LIN {X 0,Y 383.018,Z 410.271,A -85,B 0,C 180,E1 -11844.045,E2 -11844.045} C_VEL
LIN {X 0,Y 382.98,Z 410.277,A -85,B 0,C 180,E1 -11847.578,E2 -11847.578} C_VEL
LIN {X 0,Y 382.99,Z 410.275,A -85,B 0,C 180,E1 -11850.301,E2 -11850.301} C_VEL
LIN {X 0,Y 383.048,Z 410.271,A -85,B 0,C 180,E1 -11852.698,E2 -11852.698} C_VEL
LIN {X 0,Y 383.043,Z 410.273,A -85,B 0,C 180,E1 -11855.04,E2 -11855.04} C_VEL
LIN {X 0,Y 382.984,Z 410.277,A -85,B 0,C 180,E1 -11858.469,E2 -11858.469} C_VEL
LIN {X 0,Y 383.054,Z 410.266,A -85,B 0,C 180,E1 -11861.827,E2 -11861.827} C_VEL
LIN {X 0,Y 383.102,Z 410.263,A -85,B 0,C 180,E1 -11865.119,E2 -11865.119} C_VEL
LIN {X 0,Y 383.089,Z 410.265,A -85,B 0,C 180,E1 -11868.358,E2 -11868.358} C_VEL
LIN {X 0,Y 383.256,Z 410.242,A -85,B 0,C 180,E1 -11871.976,E2 -11871.976} C_VEL
LIN {X 0,Y 383.192,Z 410.255,A -85,B 0,C 180,E1 -11874.739,E2 -11874.739} C_VEL
LIN {X 0,Y 383.38,Z 410.227,A -85,B 0,C 180,E1 -11877.899,E2 -11877.899} C_VEL
LIN {X 0,Y 383.511,Z 410.211,A -85,B 0,C 180,E1 -11880.001,E2 -11880.001} C_VEL
LIN {X 0,Y 383.245,Z 410.243,A -85,B 0,C 180,E1 -11883.154,E2 -11883.154} C_VEL
LIN {X 0,Y 383.276,Z 410.244,A -85,B 0,C 180,E1 -11886.317,E2 -11886.317} C_VEL
LIN {X 0,Y 383.144,Z 410.255,A -85,B 0,C 180,E1 -11889.503,E2 -11889.503} C_VEL
LIN {X 0,Y 383.119,Z 410.259,A -85,B 0,C 180,E1 -11893.537,E2 -11893.537} C_VEL
LIN {X 0,Y 383.09,Z 410.262,A -85,B 0,C 180,E1 -11897.456,E2 -11897.456} C_VEL
LIN {X 0,Y 383.022,Z 410.272,A -85,B 0,C 180,E1 -11900.648,E2 -11900.648} C_VEL
LIN {X 0,Y 383.02,Z 410.274,A -85,B 0,C 180,E1 -11903.809,E2 -11903.809} C_VEL
LIN {X 0,Y 383.075,Z 410.271,A -85,B 0,C 180,E1 -11906.124,E2 -11906.124} C_VEL
LIN {X 0,Y 383.045,Z 410.27,A -85,B 0,C 180,E1 -11908.493,E2 -11908.493} C_VEL
LIN {X 0,Y 383.004,Z 410.275,A -85,B 0,C 180,E1 -11912.428,E2 -11912.428} C_VEL
LIN {X 0,Y 383.023,Z 410.277,A -85,B 0,C 180,E1 -11915.956,E2 -11915.956} C_VEL
LIN {X 0,Y 383.003,Z 410.279,A -85,B 0,C 180,E1 -11917.906,E2 -11917.906} C_VEL
LIN {X 0,Y 383.458,Z 413.122,A -85,B 0,C 180,E1 -11921.286,E2 -11921.286} C_VEL
LIN {X 0,Y 383.841,Z 416.038,A -85,B 0,C 180,E1 -11924.434,E2 -11924.434} C_VEL
LIN {X 0,Y 384.047,Z 419.017,A -85,B 0,C 180,E1 -11927.384,E2 -11927.384} C_VEL
LIN {X 0,Y 383.867,Z 422.184,A -85,B 0,C 180,E1 -11930.261,E2 -11930.261} C_VEL
LIN {X 0,Y 383.627,Z 425.155,A -85,B 0,C 180,E1 -11932.804,E2 -11932.804} C_VEL
LIN {X 0,Y 383.174,Z 429.849,A -85,B 0,C 180,E1 -11936.617,E2 -11936.617} C_VEL
LIN {X 0,Y 382.802,Z 433.782,A -85,B 0,C 180,E1 -11939.643,E2 -11939.643} C_VEL
LIN {X 0,Y 382.489,Z 437.86,A -85,B 0,C 180,E1 -11942.655,E2 -11942.655} C_VEL
LIN {X 0,Y 382.143,Z 442.74,A -85,B 0,C 180,E1 -11946.134,E2 -11946.134} C_VEL
LIN {X 0,Y 381.924,Z 448.017,A -85,B 0,C 180,E1 -11949.799,E2 -11949.799} C_VEL
LIN {X 0,Y 381.826,Z 450.081,A -85,B 0,C 180,E1 -11951.106,E2 -11951.106} C_VEL
LIN {X 0,Y 384.052,Z 460.663,A -85,B 0,C 180,E1 -11951.573,E2 -11951.573} C_VEL
LIN {X 0,Y 385.927,Z 471.661,A -85,B 0,C 180,E1 -11952.19,E2 -11952.19} C_VEL
LIN {X 0,Y 387.212,Z 482.447,A -85,B 0,C 180,E1 -11952.932,E2 -11952.932} C_VEL
LIN {X 0,Y 386.342,Z 494.597,A -85,B 0,C 180,E1 -11953.894,E2 -11953.894} C_VEL
LIN {X 0,Y 385.407,Z 504.894,A -85,B 0,C 180,E1 -11954.939,E2 -11954.939} C_VEL
LIN {X 0,Y 384.745,Z 512.361,A -85,B 0,C 180,E1 -11955.844,E2 -11955.844} C_VEL
LIN {X 0,Y 384.005,Z 520.647,A -85,B 0,C 180,E1 -11957.045,E2 -11957.045} C_VEL
LIN {X 0,Y 383.354,Z 526.848,A -85,B 0,C 180,E1 -11958.098,E2 -11958.098} C_VEL
LIN {X 0,Y 382.768,Z 533.386,A -85,B 0,C 180,E1 -11959.42,E2 -11959.42} C_VEL
LIN {X 0,Y 382.409,Z 537.889,A -85,B 0,C 180,E1 -11960.48,E2 -11960.48} C_VEL
LIN {X 0,Y 381.991,Z 543.381,A -85,B 0,C 180,E1 -11962.069,E2 -11962.069} C_VEL
LIN {X 0,Y 381.712,Z 547.705,A -85,B 0,C 180,E1 -11963.658,E2 -11963.658} C_VEL
LIN {X 0,Y 381.647,Z 550.072,A -85,B 0,C 180,E1 -11964.717,E2 -11964.717} C_VEL
LIN {X 0,Y 381.629,Z 551.872,A -85,B 0,C 180,E1 -11965.776,E2 -11965.776} C_VEL
LIN {X 0,Y 381.561,Z 554.315,A -85,B 0,C 180,E1 -11967.889,E2 -11967.889} C_VEL
LIN {X 0,Y 381.603,Z 554.905,A -85,B 0,C 180,E1 -11968.945,E2 -11968.945} C_VEL
LIN {X 0,Y 381.603,Z 554.905,A -85,B 0,C 180,E1 -11971.055,E2 -11971.055} C_VEL
LIN {X 0,Y 381.561,Z 554.315,A -85,B 0,C 180,E1 -11972.111,E2 -11972.111} C_VEL
LIN {X 0,Y 381.629,Z 551.872,A -85,B 0,C 180,E1 -11974.224,E2 -11974.224} C_VEL
LIN {X 0,Y 381.647,Z 550.072,A -85,B 0,C 180,E1 -11975.283,E2 -11975.283} C_VEL
LIN {X 0,Y 381.783,Z 546.464,A -85,B 0,C 180,E1 -11976.872,E2 -11976.872} C_VEL
LIN {X 0,Y 382.118,Z 541.721,A -85,B 0,C 180,E1 -11978.461,E2 -11978.461} C_VEL
LIN {X 0,Y 382.547,Z 535.697,A -85,B 0,C 180,E1 -11980.051,E2 -11980.051} C_VEL
LIN {X 0,Y 383.08,Z 529.6,A -85,B 0,C 180,E1 -11981.374,E2 -11981.374} C_VEL
LIN {X 0,Y 383.669,Z 523.9,A -85,B 0,C 180,E1 -11982.429,E2 -11982.429} C_VEL
LIN {X 0,Y 384.447,Z 515.345,A -85,B 0,C 180,E1 -11983.748,E2 -11983.748} C_VEL
LIN {X 0,Y 385.143,Z 507.162,A -85,B 0,C 180,E1 -11984.801,E2 -11984.801} C_VEL
LIN {X 0,Y 385.907,Z 498.65,A -85,B 0,C 180,E1 -11985.717,E2 -11985.717} C_VEL
LIN {X 0,Y 386.683,Z 489.935,A -85,B 0,C 180,E1 -11986.498,E2 -11986.498} C_VEL
LIN {X 0,Y 387.184,Z 482.448,A -85,B 0,C 180,E1 -11987.069,E2 -11987.069} C_VEL
LIN {X 0,Y 386.051,Z 472.502,A -85,B 0,C 180,E1 -11987.76,E2 -11987.76} C_VEL
LIN {X 0,Y 384.137,Z 461.226,A -85,B 0,C 180,E1 -11988.401,E2 -11988.401} C_VEL
LIN {X 0,Y 381.883,Z 450.583,A -85,B 0,C 180,E1 -11988.878,E2 -11988.878} C_VEL
LIN {X 0,Y 381.813,Z 449.839,A -85,B 0,C 180,E1 -11988.93,E2 -11988.93} C_VEL
LIN {X 0,Y 382.011,Z 445.986,A -85,B 0,C 180,E1 -11991.589,E2 -11991.589} C_VEL
LIN {X 0,Y 382.258,Z 441.065,A -85,B 0,C 180,E1 -11995.015,E2 -11995.015} C_VEL
LIN {X 0,Y 382.591,Z 436.226,A -85,B 0,C 180,E1 -11998.528,E2 -11998.528} C_VEL
LIN {X 0,Y 383.049,Z 431.432,A -85,B 0,C 180,E1 -12002.145,E2 -12002.145} C_VEL
LIN {X 0,Y 383.326,Z 428.263,A -85,B 0,C 180,E1 -12004.635,E2 -12004.635} C_VEL
LIN {X 0,Y 383.728,Z 424.136,A -85,B 0,C 180,E1 -12008.042,E2 -12008.042} C_VEL
LIN {X 0,Y 384,Z 420.345,A -85,B 0,C 180,E1 -12011.376,E2 -12011.376} C_VEL
LIN {X 0,Y 383.997,Z 417.514,A -85,B 0,C 180,E1 -12014.065,E2 -12014.065} C_VEL
LIN {X 0,Y 383.601,Z 414.374,A -85,B 0,C 180,E1 -12017.321,E2 -12017.321} C_VEL
LIN {X 0,Y 383.231,Z 411.685,A -85,B 0,C 180,E1 -12020.373,E2 -12020.373} C_VEL
LIN {X 0,Y 383.004,Z 410.279,A -85,B 0,C 180,E1 -12022.094,E2 -12022.094} C_VEL
LIN {X 0,Y 383.015,Z 410.279,A -85,B 0,C 180,E1 -12025.331,E2 -12025.331} C_VEL
LIN {X 0,Y 383.032,Z 410.274,A -85,B 0,C 180,E1 -12027.852,E2 -12027.852} C_VEL
LIN {X 0,Y 383.059,Z 410.27,A -85,B 0,C 180,E1 -12031.719,E2 -12031.719} C_VEL
LIN {X 0,Y 383.045,Z 410.268,A -85,B 0,C 180,E1 -12035.039,E2 -12035.039} C_VEL
LIN {X 0,Y 382.986,Z 410.276,A -85,B 0,C 180,E1 -12038.468,E2 -12038.468} C_VEL
LIN {X 0,Y 383.083,Z 410.269,A -85,B 0,C 180,E1 -12041.827,E2 -12041.827} C_VEL
LIN {X 0,Y 383.106,Z 410.261,A -85,B 0,C 180,E1 -12045.118,E2 -12045.118} C_VEL
LIN {X 0,Y 383.09,Z 410.263,A -85,B 0,C 180,E1 -12048.357,E2 -12048.357} C_VEL
LIN {X 0,Y 383.257,Z 410.244,A -85,B 0,C 180,E1 -12051.975,E2 -12051.975} C_VEL
LIN {X 0,Y 383.192,Z 410.249,A -85,B 0,C 180,E1 -12054.738,E2 -12054.738} C_VEL
LIN {X 0,Y 383.38,Z 410.228,A -85,B 0,C 180,E1 -12057.898,E2 -12057.898} C_VEL
LIN {X 0,Y 383.511,Z 410.211,A -85,B 0,C 180,E1 -12059.999,E2 -12059.999} C_VEL
LIN {X 0,Y 383.245,Z 410.246,A -85,B 0,C 180,E1 -12063.153,E2 -12063.153} C_VEL
LIN {X 0,Y 383.254,Z 410.242,A -85,B 0,C 180,E1 -12066.631,E2 -12066.631} C_VEL
LIN {X 0,Y 383.143,Z 410.26,A -85,B 0,C 180,E1 -12069.502,E2 -12069.502} C_VEL
LIN {X 0,Y 383.117,Z 410.262,A -85,B 0,C 180,E1 -12073.536,E2 -12073.536} C_VEL
LIN {X 0,Y 383.086,Z 410.266,A -85,B 0,C 180,E1 -12077.454,E2 -12077.454} C_VEL
LIN {X 0,Y 383.02,Z 410.272,A -85,B 0,C 180,E1 -12080.647,E2 -12080.647} C_VEL
LIN {X 0,Y 383.025,Z 410.271,A -85,B 0,C 180,E1 -12083.807,E2 -12083.807} C_VEL
LIN {X 0,Y 383.071,Z 410.264,A -85,B 0,C 180,E1 -12086.123,E2 -12086.123} C_VEL
LIN {X 0,Y 383.041,Z 410.27,A -85,B 0,C 180,E1 -12088.492,E2 -12088.492} C_VEL
LIN {X 0,Y 383.003,Z 410.273,A -85,B 0,C 180,E1 -12092.15,E2 -12092.15} C_VEL
LIN {X 0,Y 383.01,Z 410.276,A -85,B 0,C 180,E1 -12094.668,E2 -12094.668} C_VEL
LIN {X 0,Y 382.996,Z 410.274,A -85,B 0,C 180,E1 -12097.905,E2 -12097.905} C_VEL
LIN {X 0,Y 383.039,Z 410.27,A -85,B 0,C 180,E1 -12101.339,E2 -12101.339} C_VEL
LIN {X 0,Y 383.027,Z 410.272,A -85,B 0,C 180,E1 -12104.309,E2 -12104.309} C_VEL
LIN {X 0,Y 383.003,Z 410.274,A -85,B 0,C 180,E1 -12107.24,E2 -12107.24} C_VEL
LIN {X 0,Y 383.01,Z 410.276,A -85,B 0,C 180,E1 -12110.413,E2 -12110.413} C_VEL
LIN {X 0,Y 383.02,Z 410.272,A -85,B 0,C 180,E1 -12114.045,E2 -12114.045} C_VEL
LIN {X 0,Y 382.98,Z 410.276,A -85,B 0,C 180,E1 -12117.578,E2 -12117.578} C_VEL
LIN {X 0,Y 382.987,Z 410.279,A -85,B 0,C 180,E1 -12120.3,E2 -12120.3} C_VEL
LIN {X 0,Y 383.075,Z 410.266,A -85,B 0,C 180,E1 -12124.021,E2 -12124.021} C_VEL
LIN {X 0,Y 383.003,Z 410.273,A -85,B 0,C 180,E1 -12127.335,E2 -12127.335} C_VEL
LIN {X 0,Y 383.056,Z 410.272,A -85,B 0,C 180,E1 -12130.717,E2 -12130.717} C_VEL
LIN {X 0,Y 383.076,Z 410.27,A -85,B 0,C 180,E1 -12134.027,E2 -12134.027} C_VEL
LIN {X 0,Y 383.132,Z 410.26,A -85,B 0,C 180,E1 -12137.284,E2 -12137.284} C_VEL
LIN {X 0,Y 383.138,Z 410.274,A -85,B 0,C 180,E1 -12139.598,E2 -12139.598} C_VEL
LIN {X 0,Y 383.813,Z 412.56,A -85,B 0,C 180,E1 -12139.95,E2 -12139.95} C_VEL
LIN {X 0,Y 385.349,Z 414.562,A -85,B 0,C 180,E1 -12140.685,E2 -12140.685} C_VEL
LIN {X 0,Y 387.437,Z 415.864,A -85,B 0,C 180,E1 -12141.656,E2 -12141.656} C_VEL
LIN {X 0,Y 388.84,Z 416.565,A -85,B 0,C 180,E1 -12142.402,E2 -12142.402} C_VEL
LIN {X 0,Y 389.961,Z 418.835,A -85,B 0,C 180,E1 -12143.142,E2 -12143.142} C_VEL
LIN {X 0,Y 391.789,Z 420.997,A -85,B 0,C 180,E1 -12144.467,E2 -12144.467} C_VEL
LIN {X 0,Y 393.422,Z 422.062,A -85,B 0,C 180,E1 -12145.903,E2 -12145.903} C_VEL
LIN {X 0,Y 394.945,Z 422.432,A -85,B 0,C 180,E1 -12147.96,E2 -12147.96} C_VEL
LIN {X 0,Y 395.509,Z 422.495,A -85,B 0,C 180,E1 -12150,E2 -12150} C_VEL
LIN {X 0,Y 394.945,Z 422.432,A -85,B 0,C 180,E1 -12152.04,E2 -12152.04} C_VEL
LIN {X 0,Y 393.422,Z 422.062,A -85,B 0,C 180,E1 -12154.097,E2 -12154.097} C_VEL
LIN {X 0,Y 391.445,Z 420.702,A -85,B 0,C 180,E1 -12155.796,E2 -12155.796} C_VEL
LIN {X 0,Y 389.551,Z 418.156,A -85,B 0,C 180,E1 -12157.135,E2 -12157.135} C_VEL
LIN {X 0,Y 388.788,Z 416.4,A -85,B 0,C 180,E1 -12157.634,E2 -12157.634} C_VEL
LIN {X 0,Y 385.957,Z 415.055,A -85,B 0,C 180,E1 -12159.036,E2 -12159.036} C_VEL
LIN {X 0,Y 384.053,Z 412.977,A -85,B 0,C 180,E1 -12159.938,E2 -12159.938} C_VEL
LIN {X 0,Y 383.252,Z 410.915,A -85,B 0,C 180,E1 -12160.332,E2 -12160.332} C_VEL
LIN {X 0,Y 383.121,Z 410.262,A -85,B 0,C 180,E1 -12160.436,E2 -12160.436} C_VEL
LIN {X 0,Y 383.122,Z 410.265,A -85,B 0,C 180,E1 -12163.796,E2 -12163.796} C_VEL
LIN {X 0,Y 383.09,Z 410.267,A -85,B 0,C 180,E1 -12167.454,E2 -12167.454} C_VEL
LIN {X 0,Y 383.026,Z 410.27,A -85,B 0,C 180,E1 -12170.648,E2 -12170.648} C_VEL
LIN {X 0,Y 383.028,Z 410.274,A -85,B 0,C 180,E1 -12173.807,E2 -12173.807} C_VEL
LIN {X 0,Y 383.075,Z 410.265,A -85,B 0,C 180,E1 -12176.123,E2 -12176.123} C_VEL
LIN {X 0,Y 382.987,Z 410.279,A -85,B 0,C 180,E1 -12179.7,E2 -12179.7} C_VEL
LIN {X 0,Y 382.997,Z 410.28,A -85,B 0,C 180,E1 -12183.4,E2 -12183.4} C_VEL
LIN {X 0,Y 382.992,Z 410.272,A -85,B 0,C 180,E1 -12185.383,E2 -12185.383} C_VEL
LIN {X 0,Y 382.356,Z 410.354,A -85,B 0,C 180,E1 -12186.261,E2 -12186.261} C_VEL
LIN {X 0,Y 379.559,Z 410.706,A -85,B 0,C 180,E1 -12187.689,E2 -12187.689} C_VEL
LIN {X 0,Y 377.154,Z 411.005,A -85,B 0,C 180,E1 -12188.843,E2 -12188.843} C_VEL
LIN {X 0,Y 376.083,Z 411.138,A -85,B 0,C 180,E1 -12189.735,E2 -12189.735} C_VEL
LIN {X 0,Y 375.976,Z 411.149,A -85,B 0,C 180,E1 -12190.037,E2 -12190.037} C_VEL
LIN {X 0,Y 375.925,Z 411.156,A -85,B 0,C 180,E1 -12193.765,E2 -12193.765} C_VEL
LIN {X 0,Y 375.927,Z 411.156,A -85,B 0,C 180,E1 -12196.81,E2 -12196.81} C_VEL
LIN {X 0,Y 375.955,Z 411.152,A -85,B 0,C 180,E1 -12200.537,E2 -12200.537} C_VEL
LIN {X 0,Y 375.957,Z 411.153,A -85,B 0,C 180,E1 -12203.495,E2 -12203.495} C_VEL
LIN {X 0,Y 375.952,Z 411.151,A -85,B 0,C 180,E1 -12205.889,E2 -12205.889} C_VEL
LIN {X 0,Y 375.96,Z 411.151,A -85,B 0,C 180,E1 -12209.688,E2 -12209.688} C_VEL
LIN {X 0,Y 375.994,Z 411.146,A -85,B 0,C 180,E1 -12212.142,E2 -12212.142} C_VEL
LIN {X 0,Y 375.998,Z 411.148,A -85,B 0,C 180,E1 -12214.539,E2 -12214.539} C_VEL
LIN {X 0,Y 375.954,Z 411.151,A -85,B 0,C 180,E1 -12218.046,E2 -12218.046} C_VEL
LIN {X 0,Y 376,Z 411.146,A -85,B 0,C 180,E1 -12221.473,E2 -12221.473} C_VEL
LIN {X 0,Y 376.05,Z 411.145,A -85,B 0,C 180,E1 -12224.833,E2 -12224.833} C_VEL
LIN {X 0,Y 376.041,Z 411.141,A -85,B 0,C 180,E1 -12228.137,E2 -12228.137} C_VEL
LIN {X 0,Y 376.211,Z 411.119,A -85,B 0,C 180,E1 -12231.919,E2 -12231.919} C_VEL
LIN {X 0,Y 376.164,Z 411.131,A -85,B 0,C 180,E1 -12234.64,E2 -12234.64} C_VEL
LIN {X 0,Y 376.346,Z 411.103,A -85,B 0,C 180,E1 -12237.86,E2 -12237.86} C_VEL
LIN {X 0,Y 376.481,Z 411.087,A -85,B 0,C 180,E1 -12240.001,E2 -12240.001} C_VEL
LIN {X 0,Y 376.183,Z 411.123,A -85,B 0,C 180,E1 -12243.214,E2 -12243.214} C_VEL
LIN {X 0,Y 376.234,Z 411.123,A -85,B 0,C 180,E1 -12246.436,E2 -12246.436} C_VEL
LIN {X 0,Y 376.112,Z 411.132,A -85,B 0,C 180,E1 -12249.682,E2 -12249.682} C_VEL
LIN {X 0,Y 376.083,Z 411.136,A -85,B 0,C 180,E1 -12253.658,E2 -12253.658} C_VEL
LIN {X 0,Y 376.039,Z 411.141,A -85,B 0,C 180,E1 -12257.609,E2 -12257.609} C_VEL
LIN {X 0,Y 375.973,Z 411.149,A -85,B 0,C 180,E1 -12260.833,E2 -12260.833} C_VEL
LIN {X 0,Y 375.984,Z 411.152,A -85,B 0,C 180,E1 -12264.283,E2 -12264.283} C_VEL
LIN {X 0,Y 376.015,Z 411.145,A -85,B 0,C 180,E1 -12266.653,E2 -12266.653} C_VEL
LIN {X 0,Y 375.972,Z 411.149,A -85,B 0,C 180,E1 -12269.08,E2 -12269.08} C_VEL
LIN {X 0,Y 375.954,Z 411.151,A -85,B 0,C 180,E1 -12272.829,E2 -12272.829} C_VEL
LIN {X 0,Y 375.955,Z 411.153,A -85,B 0,C 180,E1 -12275.416,E2 -12275.416} C_VEL
LIN {X 0,Y 375.952,Z 411.156,A -85,B 0,C 180,E1 -12276.742,E2 -12276.742} C_VEL
LIN {X 0,Y 376.032,Z 411.717,A -85,B 0,C 180,E1 -12278.283,E2 -12278.283} C_VEL
LIN {X 0,Y 376.483,Z 414.575,A -85,B 0,C 180,E1 -12281.696,E2 -12281.696} C_VEL
LIN {X 0,Y 376.885,Z 417.758,A -85,B 0,C 180,E1 -12285.122,E2 -12285.122} C_VEL
LIN {X 0,Y 376.979,Z 420.516,A -85,B 0,C 180,E1 -12287.846,E2 -12287.846} C_VEL
LIN {X 0,Y 376.791,Z 423.56,A -85,B 0,C 180,E1 -12290.642,E2 -12290.642} C_VEL
LIN {X 0,Y 376.516,Z 426.717,A -85,B 0,C 180,E1 -12293.383,E2 -12293.383} C_VEL
LIN {X 0,Y 376.062,Z 431.355,A -85,B 0,C 180,E1 -12297.183,E2 -12297.183} C_VEL
LIN {X 0,Y 375.746,Z 434.529,A -85,B 0,C 180,E1 -12299.669,E2 -12299.669} C_VEL
LIN {X 0,Y 375.33,Z 439.35,A -85,B 0,C 180,E1 -12303.296,E2 -12303.296} C_VEL
LIN {X 0,Y 375.036,Z 444.211,A -85,B 0,C 180,E1 -12306.826,E2 -12306.826} C_VEL
LIN {X 0,Y 374.782,Z 449.874,A -85,B 0,C 180,E1 -12310.737,E2 -12310.737} C_VEL
LIN {X 0,Y 376.999,Z 460.456,A -85,B 0,C 180,E1 -12311.216,E2 -12311.216} C_VEL
LIN {X 0,Y 378.729,Z 470.398,A -85,B 0,C 180,E1 -12311.783,E2 -12311.783} C_VEL
LIN {X 0,Y 379.965,Z 479.75,A -85,B 0,C 180,E1 -12312.425,E2 -12312.425} C_VEL
LIN {X 0,Y 380.278,Z 484.84,A -85,B 0,C 180,E1 -12312.801,E2 -12312.801} C_VEL
LIN {X 0,Y 379.366,Z 495.751,A -85,B 0,C 180,E1 -12313.728,E2 -12313.728} C_VEL
LIN {X 0,Y 378.534,Z 504.696,A -85,B 0,C 180,E1 -12314.659,E2 -12314.659} C_VEL
LIN {X 0,Y 377.812,Z 512.513,A -85,B 0,C 180,E1 -12315.629,E2 -12315.629} C_VEL
LIN {X 0,Y 377.072,Z 520.449,A -85,B 0,C 180,E1 -12316.802,E2 -12316.802} C_VEL
LIN {X 0,Y 376.396,Z 526.65,A -85,B 0,C 180,E1 -12317.875,E2 -12317.875} C_VEL
LIN {X 0,Y 375.745,Z 533.188,A -85,B 0,C 180,E1 -12319.22,E2 -12319.22} C_VEL
LIN {X 0,Y 375.372,Z 537.691,A -85,B 0,C 180,E1 -12320.299,E2 -12320.299} C_VEL
LIN {X 0,Y 374.925,Z 543.183,A -85,B 0,C 180,E1 -12321.918,E2 -12321.918} C_VEL
LIN {X 0,Y 374.633,Z 547.507,A -85,B 0,C 180,E1 -12323.537,E2 -12323.537} C_VEL
LIN {X 0,Y 374.555,Z 549.874,A -85,B 0,C 180,E1 -12324.617,E2 -12324.617} C_VEL
LIN {X 0,Y 374.555,Z 551.675,A -85,B 0,C 180,E1 -12325.696,E2 -12325.696} C_VEL
LIN {X 0,Y 374.46,Z 554.118,A -85,B 0,C 180,E1 -12327.849,E2 -12327.849} C_VEL
LIN {X 0,Y 374.503,Z 554.708,A -85,B 0,C 180,E1 -12328.925,E2 -12328.925} C_VEL
LIN {X 0,Y 374.503,Z 554.708,A -85,B 0,C 180,E1 -12331.075,E2 -12331.075} C_VEL
LIN {X 0,Y 374.46,Z 554.118,A -85,B 0,C 180,E1 -12332.151,E2 -12332.151} C_VEL
LIN {X 0,Y 374.555,Z 551.675,A -85,B 0,C 180,E1 -12334.304,E2 -12334.304} C_VEL
LIN {X 0,Y 374.585,Z 548.397,A -85,B 0,C 180,E1 -12336.068,E2 -12336.068} C_VEL
LIN {X 0,Y 374.809,Z 544.736,A -85,B 0,C 180,E1 -12337.542,E2 -12337.542} C_VEL
LIN {X 0,Y 375.221,Z 539.607,A -85,B 0,C 180,E1 -12339.161,E2 -12339.161} C_VEL
LIN {X 0,Y 375.662,Z 534.344,A -85,B 0,C 180,E1 -12340.51,E2 -12340.51} C_VEL
LIN {X 0,Y 376.226,Z 528.026,A -85,B 0,C 180,E1 -12341.857,E2 -12341.857} C_VEL
LIN {X 0,Y 376.894,Z 522.076,A -85,B 0,C 180,E1 -12342.93,E2 -12342.93} C_VEL
LIN {X 0,Y 377.655,Z 513.898,A -85,B 0,C 180,E1 -12344.179,E2 -12344.179} C_VEL
LIN {X 0,Y 378.36,Z 505.829,A -85,B 0,C 180,E1 -12345.21,E2 -12345.21} C_VEL
LIN {X 0,Y 379.187,Z 497.101,A -85,B 0,C 180,E1 -12346.141,E2 -12346.141} C_VEL
LIN {X 0,Y 380.025,Z 488.106,A -85,B 0,C 180,E1 -12346.934,E2 -12346.934} C_VEL
LIN {X 0,Y 380.264,Z 482.387,A -85,B 0,C 180,E1 -12347.38,E2 -12347.38} C_VEL
LIN {X 0,Y 379.091,Z 472.83,A -85,B 0,C 180,E1 -12348.068,E2 -12348.068} C_VEL
LIN {X 0,Y 377.105,Z 460.921,A -85,B 0,C 180,E1 -12348.76,E2 -12348.76} C_VEL
LIN {X 0,Y 374.839,Z 450.544,A -85,B 0,C 180,E1 -12349.242,E2 -12349.242} C_VEL
LIN {X 0,Y 374.781,Z 449.672,A -85,B 0,C 180,E1 -12349.299,E2 -12349.299} C_VEL
LIN {X 0,Y 375.037,Z 444.204,A -85,B 0,C 180,E1 -12353.174,E2 -12353.174} C_VEL
LIN {X 0,Y 375.32,Z 439.341,A -85,B 0,C 180,E1 -12356.705,E2 -12356.705} C_VEL
LIN {X 0,Y 375.747,Z 434.527,A -85,B 0,C 180,E1 -12360.331,E2 -12360.331} C_VEL
LIN {X 0,Y 376.063,Z 431.35,A -85,B 0,C 180,E1 -12362.817,E2 -12362.817} C_VEL
LIN {X 0,Y 376.516,Z 426.714,A -85,B 0,C 180,E1 -12366.617,E2 -12366.617} C_VEL
LIN {X 0,Y 376.791,Z 423.554,A -85,B 0,C 180,E1 -12369.358,E2 -12369.358} C_VEL
LIN {X 0,Y 376.993,Z 420.506,A -85,B 0,C 180,E1 -12372.152,E2 -12372.152} C_VEL
LIN {X 0,Y 376.85,Z 417.5,A -85,B 0,C 180,E1 -12375.126,E2 -12375.126} C_VEL
LIN {X 0,Y 376.481,Z 414.575,A -85,B 0,C 180,E1 -12378.304,E2 -12378.304} C_VEL
LIN {X 0,Y 376.011,Z 411.559,A -85,B 0,C 180,E1 -12381.916,E2 -12381.916} C_VEL
LIN {X 0,Y 375.962,Z 411.155,A -85,B 0,C 180,E1 -12383.494,E2 -12383.494} C_VEL
LIN {X 0,Y 375.96,Z 411.157,A -85,B 0,C 180,E1 -12385.888,E2 -12385.888} C_VEL
LIN {X 0,Y 375.965,Z 411.153,A -85,B 0,C 180,E1 -12389.687,E2 -12389.687} C_VEL
LIN {X 0,Y 375.998,Z 411.15,A -85,B 0,C 180,E1 -12392.141,E2 -12392.141} C_VEL
LIN {X 0,Y 376,Z 411.146,A -85,B 0,C 180,E1 -12394.538,E2 -12394.538} C_VEL
LIN {X 0,Y 375.952,Z 411.155,A -85,B 0,C 180,E1 -12398.044,E2 -12398.044} C_VEL
LIN {X 0,Y 376.018,Z 411.146,A -85,B 0,C 180,E1 -12401.473,E2 -12401.473} C_VEL
LIN {X 0,Y 376.054,Z 411.138,A -85,B 0,C 180,E1 -12404.832,E2 -12404.832} C_VEL
LIN {X 0,Y 376.042,Z 411.142,A -85,B 0,C 180,E1 -12408.136,E2 -12408.136} C_VEL
LIN {X 0,Y 376.212,Z 411.122,A -85,B 0,C 180,E1 -12411.918,E2 -12411.918} C_VEL
LIN {X 0,Y 376.164,Z 411.125,A -85,B 0,C 180,E1 -12414.639,E2 -12414.639} C_VEL
LIN {X 0,Y 376.346,Z 411.105,A -85,B 0,C 180,E1 -12417.859,E2 -12417.859} C_VEL
LIN {X 0,Y 376.481,Z 411.087,A -85,B 0,C 180,E1 -12419.999,E2 -12419.999} C_VEL
LIN {X 0,Y 376.183,Z 411.127,A -85,B 0,C 180,E1 -12423.212,E2 -12423.212} C_VEL
LIN {X 0,Y 376.219,Z 411.118,A -85,B 0,C 180,E1 -12426.619,E2 -12426.619} C_VEL
LIN {X 0,Y 376.111,Z 411.134,A -85,B 0,C 180,E1 -12429.681,E2 -12429.681} C_VEL
LIN {X 0,Y 376.081,Z 411.137,A -85,B 0,C 180,E1 -12433.657,E2 -12433.657} C_VEL
LIN {X 0,Y 376.034,Z 411.143,A -85,B 0,C 180,E1 -12437.606,E2 -12437.606} C_VEL
LIN {X 0,Y 375.97,Z 411.152,A -85,B 0,C 180,E1 -12440.832,E2 -12440.832} C_VEL
LIN {X 0,Y 375.985,Z 411.147,A -85,B 0,C 180,E1 -12444.281,E2 -12444.281} C_VEL
LIN {X 0,Y 376.011,Z 411.146,A -85,B 0,C 180,E1 -12446.652,E2 -12446.652} C_VEL
LIN {X 0,Y 375.968,Z 411.155,A -85,B 0,C 180,E1 -12449.079,E2 -12449.079} C_VEL
LIN {X 0,Y 375.941,Z 411.158,A -85,B 0,C 180,E1 -12452.828,E2 -12452.828} C_VEL
LIN {X 0,Y 375.95,Z 411.153,A -85,B 0,C 180,E1 -12455.415,E2 -12455.415} C_VEL
LIN {X 0,Y 375.97,Z 411.15,A -85,B 0,C 180,E1 -12458.271,E2 -12458.271} C_VEL
LIN {X 0,Y 375.982,Z 411.148,A -85,B 0,C 180,E1 -12461.61,E2 -12461.61} C_VEL
LIN {X 0,Y 375.963,Z 411.151,A -85,B 0,C 180,E1 -12465.262,E2 -12465.262} C_VEL
LIN {X 0,Y 375.935,Z 411.155,A -85,B 0,C 180,E1 -12469.133,E2 -12469.133} C_VEL
LIN {X 0,Y 375.96,Z 411.151,A -85,B 0,C 180,E1 -12471.912,E2 -12471.912} C_VEL
LIN {X 0,Y 375.974,Z 411.149,A -85,B 0,C 180,E1 -12475.333,E2 -12475.333} C_VEL
LIN {X 0,Y 375.952,Z 411.157,A -85,B 0,C 180,E1 -12478.438,E2 -12478.438} C_VEL
LIN {X 0,Y 375.978,Z 411.151,A -85,B 0,C 180,E1 -12482.141,E2 -12482.141} C_VEL
LIN {X 0,Y 376.002,Z 411.15,A -85,B 0,C 180,E1 -12484.539,E2 -12484.539} C_VEL
LIN {X 0,Y 375.958,Z 411.154,A -85,B 0,C 180,E1 -12488.046,E2 -12488.046} C_VEL
LIN {X 0,Y 376.019,Z 411.147,A -85,B 0,C 180,E1 -12491.474,E2 -12491.474} C_VEL
LIN {X 0,Y 376.054,Z 411.143,A -85,B 0,C 180,E1 -12494.833,E2 -12494.833} C_VEL
LIN {X 0,Y 376.117,Z 411.317,A -85,B 0,C 180,E1 -12497.317,E2 -12497.317} C_VEL
LIN {X 0,Y 376.87,Z 413.647,A -85,B 0,C 180,E1 -12497.651,E2 -12497.651} C_VEL
LIN {X 0,Y 378.821,Z 415.935,A -85,B 0,C 180,E1 -12498.361,E2 -12498.361} C_VEL
LIN {X 0,Y 381.132,Z 417.187,A -85,B 0,C 180,E1 -12499.206,E2 -12499.206} C_VEL
LIN {X 0,Y 382.48,Z 419.777,A -85,B 0,C 180,E1 -12499.813,E2 -12499.813} C_VEL
LIN {X 0,Y 384.674,Z 421.95,A -85,B 0,C 180,E1 -12500.801,E2 -12500.801} C_VEL
LIN {X 0,Y 387.406,Z 423.442,A -85,B 0,C 180,E1 -12502.125,E2 -12502.125} C_VEL
LIN {X 0,Y 388.935,Z 426,A -85,B 0,C 180,E1 -12503.079,E2 -12503.079} C_VEL
LIN {X 0,Y 390.889,Z 428.079,A -85,B 0,C 180,E1 -12504.454,E2 -12504.454} C_VEL
LIN {X 0,Y 392.534,Z 429.093,A -85,B 0,C 180,E1 -12505.893,E2 -12505.893} C_VEL
LIN {X 0,Y 394.082,Z 429.478,A -85,B 0,C 180,E1 -12507.956,E2 -12507.956} C_VEL
LIN {X 0,Y 394.645,Z 429.534,A -85,B 0,C 180,E1 -12510,E2 -12510} C_VEL
LIN {X 0,Y 394.082,Z 429.478,A -85,B 0,C 180,E1 -12512.044,E2 -12512.044} C_VEL
LIN {X 0,Y 392.534,Z 429.095,A -85,B 0,C 180,E1 -12514.107,E2 -12514.107} C_VEL
LIN {X 0,Y 390.528,Z 427.799,A -85,B 0,C 180,E1 -12515.81,E2 -12515.81} C_VEL
LIN {X 0,Y 388.395,Z 425.214,A -85,B 0,C 180,E1 -12517.277,E2 -12517.277} C_VEL
LIN {X 0,Y 387.179,Z 423.139,A -85,B 0,C 180,E1 -12518.007,E2 -12518.007} C_VEL
LIN {X 0,Y 384.525,Z 421.838,A -85,B 0,C 180,E1 -12519.267,E2 -12519.267} C_VEL
LIN {X 0,Y 382.316,Z 419.545,A -85,B 0,C 180,E1 -12520.258,E2 -12520.258} C_VEL
LIN {X 0,Y 380.992,Z 417.036,A -85,B 0,C 180,E1 -12520.852,E2 -12520.852} C_VEL
LIN {X 0,Y 378.583,Z 415.749,A -85,B 0,C 180,E1 -12521.721,E2 -12521.721} C_VEL
LIN {X 0,Y 376.776,Z 413.476,A -85,B 0,C 180,E1 -12522.386,E2 -12522.386} C_VEL
LIN {X 0,Y 376.085,Z 411.139,A -85,B 0,C 180,E1 -12522.752,E2 -12522.752} C_VEL
LIN {X 0,Y 376.025,Z 411.148,A -85,B 0,C 180,E1 -12526.281,E2 -12526.281} C_VEL
LIN {X 0,Y 375.994,Z 411.153,A -85,B 0,C 180,E1 -12529.66,E2 -12529.66} C_VEL
LIN {X 0,Y 375.991,Z 411.152,A -85,B 0,C 180,E1 -12533.667,E2 -12533.667} C_VEL
LIN {X 0,Y 376.014,Z 411.143,A -85,B 0,C 180,E1 -12536.652,E2 -12536.652} C_VEL
LIN {X 0,Y 375.959,Z 411.15,A -85,B 0,C 180,E1 -12540.312,E2 -12540.312} C_VEL
LIN {X 0,Y 375.954,Z 411.152,A -85,B 0,C 180,E1 -12544.111,E2 -12544.111} C_VEL
LIN {X 0,Y 375.948,Z 411.152,A -85,B 0,C 180,E1 -12546.741,E2 -12546.741} C_VEL
LIN {X 0,Y 375.976,Z 411.149,A -85,B 0,C 180,E1 -12550.037,E2 -12550.037} C_VEL
LIN {X 0,Y 375.243,Z 411.244,A -85,B 0,C 180,E1 -12550.931,E2 -12550.931} C_VEL
LIN {X 0,Y 372.336,Z 411.602,A -85,B 0,C 180,E1 -12552.383,E2 -12552.383} C_VEL
LIN {X 0,Y 369.939,Z 411.904,A -85,B 0,C 180,E1 -12553.557,E2 -12553.557} C_VEL
LIN {X 0,Y 368.955,Z 412.023,A -85,B 0,C 180,E1 -12554.466,E2 -12554.466} C_VEL
LIN {X 0,Y 368.897,Z 412.032,A -85,B 0,C 180,E1 -12554.773,E2 -12554.773} C_VEL
LIN {X 0,Y 368.875,Z 412.033,A -85,B 0,C 180,E1 -12558.177,E2 -12558.177} C_VEL
LIN {X 0,Y 368.902,Z 412.034,A -85,B 0,C 180,E1 -12561.359,E2 -12561.359} C_VEL
LIN {X 0,Y 368.929,Z 412.032,A -85,B 0,C 180,E1 -12565.146,E2 -12565.146} C_VEL
LIN {X 0,Y 368.921,Z 412.034,A -85,B 0,C 180,E1 -12569.047,E2 -12569.047} C_VEL
LIN {X 0,Y 368.979,Z 412.021,A -85,B 0,C 180,E1 -12571.565,E2 -12571.565} C_VEL
LIN {X 0,Y 368.949,Z 412.027,A -85,B 0,C 180,E1 -12575.225,E2 -12575.225} C_VEL
LIN {X 0,Y 368.929,Z 412.031,A -85,B 0,C 180,E1 -12578.974,E2 -12578.974} C_VEL
LIN {X 0,Y 368.982,Z 412.021,A -85,B 0,C 180,E1 -12582.257,E2 -12582.257} C_VEL
LIN {X 0,Y 369.029,Z 412.015,A -85,B 0,C 180,E1 -12586.228,E2 -12586.228} C_VEL
LIN {X 0,Y 369.059,Z 412.011,A -85,B 0,C 180,E1 -12590.132,E2 -12590.132} C_VEL
LIN {X 0,Y 369.194,Z 411.993,A -85,B 0,C 180,E1 -12593.442,E2 -12593.442} C_VEL
LIN {X 0,Y 369.311,Z 411.979,A -85,B 0,C 180,E1 -12597.819,E2 -12597.819} C_VEL
LIN {X 0,Y 369.45,Z 411.962,A -85,B 0,C 180,E1 -12600.001,E2 -12600.001} C_VEL
LIN {X 0,Y 369.311,Z 411.982,A -85,B 0,C 180,E1 -12602.182,E2 -12602.182} C_VEL
LIN {X 0,Y 369.194,Z 411.998,A -85,B 0,C 180,E1 -12606.559,E2 -12606.559} C_VEL
LIN {X 0,Y 369.06,Z 412.011,A -85,B 0,C 180,E1 -12609.869,E2 -12609.869} C_VEL
LIN {X 0,Y 369.03,Z 412.015,A -85,B 0,C 180,E1 -12613.773,E2 -12613.773} C_VEL
LIN {X 0,Y 368.995,Z 412.02,A -85,B 0,C 180,E1 -12617.769,E2 -12617.769} C_VEL
LIN {X 0,Y 368.904,Z 412.029,A -85,B 0,C 180,E1 -12621.222,E2 -12621.222} C_VEL
LIN {X 0,Y 368.95,Z 412.024,A -85,B 0,C 180,E1 -12624.777,E2 -12624.777} C_VEL
LIN {X 0,Y 368.966,Z 412.021,A -85,B 0,C 180,E1 -12627.204,E2 -12627.204} C_VEL
LIN {X 0,Y 368.919,Z 412.03,A -85,B 0,C 180,E1 -12629.691,E2 -12629.691} C_VEL
LIN {X 0,Y 368.898,Z 412.032,A -85,B 0,C 180,E1 -12633.539,E2 -12633.539} C_VEL
LIN {X 0,Y 368.9,Z 412.035,A -85,B 0,C 180,E1 -12636.857,E2 -12636.857} C_VEL
LIN {X 0,Y 369.117,Z 413.367,A -85,B 0,C 180,E1 -12638.927,E2 -12638.927} C_VEL
LIN {X 0,Y 369.538,Z 416.054,A -85,B 0,C 180,E1 -12642.124,E2 -12642.124} C_VEL
LIN {X 0,Y 369.87,Z 418.989,A -85,B 0,C 180,E1 -12645.329,E2 -12645.329} C_VEL
LIN {X 0,Y 369.926,Z 421.994,A -85,B 0,C 180,E1 -12648.323,E2 -12648.323} C_VEL
LIN {X 0,Y 369.704,Z 425.114,A -85,B 0,C 180,E1 -12651.207,E2 -12651.207} C_VEL
LIN {X 0,Y 369.385,Z 428.142,A -85,B 0,C 180,E1 -12653.857,E2 -12653.857} C_VEL
LIN {X 0,Y 369.014,Z 431.822,A -85,B 0,C 180,E1 -12656.93,E2 -12656.93} C_VEL
LIN {X 0,Y 368.572,Z 436.028,A -85,B 0,C 180,E1 -12660.28,E2 -12660.28} C_VEL
LIN {X 0,Y 368.19,Z 440.843,A -85,B 0,C 180,E1 -12663.959,E2 -12663.959} C_VEL
LIN {X 0,Y 367.874,Z 445.708,A -85,B 0,C 180,E1 -12667.538,E2 -12667.538} C_VEL
LIN {X 0,Y 367.703,Z 449.665,A -85,B 0,C 180,E1 -12670.351,E2 -12670.351} C_VEL
LIN {X 0,Y 369.845,Z 459.748,A -85,B 0,C 180,E1 -12670.818,E2 -12670.818} C_VEL
LIN {X 0,Y 371.599,Z 469.263,A -85,B 0,C 180,E1 -12671.369,E2 -12671.369} C_VEL
LIN {X 0,Y 372.937,Z 478.557,A -85,B 0,C 180,E1 -12672.013,E2 -12672.013} C_VEL
LIN {X 0,Y 373.474,Z 484.642,A -85,B 0,C 180,E1 -12672.478,E2 -12672.478} C_VEL
LIN {X 0,Y 372.543,Z 495.554,A -85,B 0,C 180,E1 -12673.422,E2 -12673.422} C_VEL
LIN {X 0,Y 371.666,Z 504.499,A -85,B 0,C 180,E1 -12674.368,E2 -12674.368} C_VEL
LIN {X 0,Y 370.836,Z 513.088,A -85,B 0,C 180,E1 -12675.466,E2 -12675.466} C_VEL
LIN {X 0,Y 370.127,Z 520.251,A -85,B 0,C 180,E1 -12676.55,E2 -12676.55} C_VEL
LIN {X 0,Y 369.446,Z 526.453,A -85,B 0,C 180,E1 -12677.643,E2 -12677.643} C_VEL
LIN {X 0,Y 368.73,Z 532.989,A -85,B 0,C 180,E1 -12679.012,E2 -12679.012} C_VEL
LIN {X 0,Y 368.321,Z 537.492,A -85,B 0,C 180,E1 -12680.112,E2 -12680.112} C_VEL
LIN {X 0,Y 367.878,Z 542.985,A -85,B 0,C 180,E1 -12681.762,E2 -12681.762} C_VEL
LIN {X 0,Y 367.566,Z 547.31,A -85,B 0,C 180,E1 -12683.413,E2 -12683.413} C_VEL
LIN {X 0,Y 367.467,Z 549.677,A -85,B 0,C 180,E1 -12684.513,E2 -12684.513} C_VEL
LIN {X 0,Y 367.46,Z 551.477,A -85,B 0,C 180,E1 -12685.612,E2 -12685.612} C_VEL
LIN {X 0,Y 367.361,Z 553.921,A -85,B 0,C 180,E1 -12687.807,E2 -12687.807} C_VEL
LIN {X 0,Y 367.404,Z 554.511,A -85,B 0,C 180,E1 -12688.904,E2 -12688.904} C_VEL
LIN {X 0,Y 367.404,Z 554.511,A -85,B 0,C 180,E1 -12691.096,E2 -12691.096} C_VEL
LIN {X 0,Y 367.361,Z 553.921,A -85,B 0,C 180,E1 -12692.193,E2 -12692.193} C_VEL
LIN {X 0,Y 367.46,Z 551.477,A -85,B 0,C 180,E1 -12694.388,E2 -12694.388} C_VEL
LIN {X 0,Y 367.483,Z 548.573,A -85,B 0,C 180,E1 -12696.016,E2 -12696.016} C_VEL
LIN {X 0,Y 367.736,Z 544.538,A -85,B 0,C 180,E1 -12697.688,E2 -12697.688} C_VEL
LIN {X 0,Y 368.166,Z 539.409,A -85,B 0,C 180,E1 -12699.338,E2 -12699.338} C_VEL
LIN {X 0,Y 368.628,Z 534.146,A -85,B 0,C 180,E1 -12700.713,E2 -12700.713} C_VEL
LIN {X 0,Y 369.269,Z 527.828,A -85,B 0,C 180,E1 -12702.084,E2 -12702.084} C_VEL
LIN {X 0,Y 369.949,Z 521.878,A -85,B 0,C 180,E1 -12703.177,E2 -12703.177} C_VEL
LIN {X 0,Y 370.617,Z 514.949,A -85,B 0,C 180,E1 -12704.271,E2 -12704.271} C_VEL
LIN {X 0,Y 371.368,Z 506.766,A -85,B 0,C 180,E1 -12705.363,E2 -12705.363} C_VEL
LIN {X 0,Y 372.222,Z 498.255,A -85,B 0,C 180,E1 -12706.311,E2 -12706.311} C_VEL
LIN {X 0,Y 373.094,Z 489.541,A -85,B 0,C 180,E1 -12707.117,E2 -12707.117} C_VEL
LIN {X 0,Y 373.435,Z 483.548,A -85,B 0,C 180,E1 -12707.612,E2 -12707.612} C_VEL
LIN {X 0,Y 371.92,Z 471.488,A -85,B 0,C 180,E1 -12708.492,E2 -12708.492} C_VEL
LIN {X 0,Y 370.061,Z 460.66,A -85,B 0,C 180,E1 -12709.133,E2 -12709.133} C_VEL
LIN {X 0,Y 367.709,Z 449.507,A -85,B 0,C 180,E1 -12709.682,E2 -12709.682} C_VEL
LIN {X 0,Y 367.971,Z 444.059,A -85,B 0,C 180,E1 -12713.645,E2 -12713.645} C_VEL
LIN {X 0,Y 368.318,Z 439.221,A -85,B 0,C 180,E1 -12717.254,E2 -12717.254} C_VEL
LIN {X 0,Y 368.774,Z 434.422,A -85,B 0,C 180,E1 -12720.967,E2 -12720.967} C_VEL
LIN {X 0,Y 369.239,Z 429.694,A -85,B 0,C 180,E1 -12724.82,E2 -12724.82} C_VEL
LIN {X 0,Y 369.546,Z 426.587,A -85,B 0,C 180,E1 -12727.485,E2 -12727.485} C_VEL
LIN {X 0,Y 369.851,Z 423.207,A -85,B 0,C 180,E1 -12730.527,E2 -12730.527} C_VEL
LIN {X 0,Y 369.969,Z 420.475,A -85,B 0,C 180,E1 -12733.145,E2 -12733.145} C_VEL
LIN {X 0,Y 369.705,Z 417.517,A -85,B 0,C 180,E1 -12736.249,E2 -12736.249} C_VEL
LIN {X 0,Y 369.278,Z 414.501,A -85,B 0,C 180,E1 -12739.678,E2 -12739.678} C_VEL
LIN {X 0,Y 368.945,Z 412.293,A -85,B 0,C 180,E1 -12742.441,E2 -12742.441} C_VEL
LIN {X 0,Y 368.933,Z 412.033,A -85,B 0,C 180,E1 -12745.145,E2 -12745.145} C_VEL
LIN {X 0,Y 368.925,Z 412.026,A -85,B 0,C 180,E1 -12749.045,E2 -12749.045} C_VEL
LIN {X 0,Y 368.982,Z 412.022,A -85,B 0,C 180,E1 -12751.564,E2 -12751.564} C_VEL
LIN {X 0,Y 368.995,Z 412.023,A -85,B 0,C 180,E1 -12754.019,E2 -12754.019} C_VEL
LIN {X 0,Y 368.919,Z 412.031,A -85,B 0,C 180,E1 -12757.603,E2 -12757.603} C_VEL
LIN {X 0,Y 368.961,Z 412.023,A -85,B 0,C 180,E1 -12761.105,E2 -12761.105} C_VEL
LIN {X 0,Y 368.994,Z 412.018,A -85,B 0,C 180,E1 -12764.534,E2 -12764.534} C_VEL
LIN {X 0,Y 368.998,Z 412.021,A -85,B 0,C 180,E1 -12767.906,E2 -12767.906} C_VEL
LIN {X 0,Y 369.159,Z 412.001,A -85,B 0,C 180,E1 -12771.868,E2 -12771.868} C_VEL
LIN {X 0,Y 369.136,Z 412,A -85,B 0,C 180,E1 -12774.537,E2 -12774.537} C_VEL
LIN {X 0,Y 369.311,Z 411.982,A -85,B 0,C 180,E1 -12777.818,E2 -12777.818} C_VEL
LIN {X 0,Y 369.45,Z 411.962,A -85,B 0,C 180,E1 -12779.999,E2 -12779.999} C_VEL
LIN {X 0,Y 369.311,Z 411.979,A -85,B 0,C 180,E1 -12782.181,E2 -12782.181} C_VEL
LIN {X 0,Y 369.189,Z 411.994,A -85,B 0,C 180,E1 -12786.604,E2 -12786.604} C_VEL
LIN {X 0,Y 369.059,Z 412.011,A -85,B 0,C 180,E1 -12789.868,E2 -12789.868} C_VEL
LIN {X 0,Y 369.029,Z 412.015,A -85,B 0,C 180,E1 -12793.772,E2 -12793.772} C_VEL
LIN {X 0,Y 368.993,Z 412.019,A -85,B 0,C 180,E1 -12797.768,E2 -12797.768} C_VEL
LIN {X 0,Y 368.921,Z 412.033,A -85,B 0,C 180,E1 -12801.219,E2 -12801.219} C_VEL
LIN {X 0,Y 368.949,Z 412.027,A -85,B 0,C 180,E1 -12804.775,E2 -12804.775} C_VEL
LIN {X 0,Y 368.979,Z 412.021,A -85,B 0,C 180,E1 -12808.435,E2 -12808.435} C_VEL
LIN {X 0,Y 368.891,Z 412.031,A -85,B 0,C 180,E1 -12812.238,E2 -12812.238} C_VEL
LIN {X 0,Y 368.921,Z 412.032,A -85,B 0,C 180,E1 -12815.002,E2 -12815.002} C_VEL
LIN {X 0,Y 368.906,Z 412.033,A -85,B 0,C 180,E1 -12818.641,E2 -12818.641} C_VEL
LIN {X 0,Y 368.934,Z 412.026,A -85,B 0,C 180,E1 -12822.02,E2 -12822.02} C_VEL
LIN {X 0,Y 368.917,Z 412.029,A -85,B 0,C 180,E1 -12825.183,E2 -12825.183} C_VEL
LIN {X 0,Y 368.877,Z 412.034,A -85,B 0,C 180,E1 -12828.178,E2 -12828.178} C_VEL
LIN {X 0,Y 368.904,Z 412.03,A -85,B 0,C 180,E1 -12831.36,E2 -12831.36} C_VEL
LIN {X 0,Y 368.93,Z 412.027,A -85,B 0,C 180,E1 -12835.147,E2 -12835.147} C_VEL
LIN {X 0,Y 368.923,Z 412.028,A -85,B 0,C 180,E1 -12839.047,E2 -12839.047} C_VEL
LIN {X 0,Y 368.958,Z 412.025,A -85,B 0,C 180,E1 -12842.797,E2 -12842.797} C_VEL
LIN {X 0,Y 368.94,Z 412.028,A -85,B 0,C 180,E1 -12846.113,E2 -12846.113} C_VEL
LIN {X 0,Y 368.932,Z 412.029,A -85,B 0,C 180,E1 -12849.947,E2 -12849.947} C_VEL
LIN {X 0,Y 368.971,Z 412.026,A -85,B 0,C 180,E1 -12853.399,E2 -12853.399} C_VEL
LIN {X 0,Y 369,Z 412.044,A -85,B 0,C 180,E1 -12855.418,E2 -12855.418} C_VEL
LIN {X 0,Y 369.846,Z 414.591,A -85,B 0,C 180,E1 -12855.723,E2 -12855.723} C_VEL
LIN {X 0,Y 371.533,Z 416.597,A -85,B 0,C 180,E1 -12856.237,E2 -12856.237} C_VEL
LIN {X 0,Y 373.68,Z 417.939,A -85,B 0,C 180,E1 -12856.887,E2 -12856.887} C_VEL
LIN {X 0,Y 375.293,Z 420.76,A -85,B 0,C 180,E1 -12857.46,E2 -12857.46} C_VEL
LIN {X 0,Y 377.838,Z 423.125,A -85,B 0,C 180,E1 -12858.358,E2 -12858.358} C_VEL
LIN {X 0,Y 379.349,Z 424.068,A -85,B 0,C 180,E1 -12858.896,E2 -12858.896} C_VEL
LIN {X 0,Y 381.256,Z 426.95,A -85,B 0,C 180,E1 -12859.713,E2 -12859.713} C_VEL
LIN {X 0,Y 384.014,Z 429.233,A -85,B 0,C 180,E1 -12860.918,E2 -12860.918} C_VEL
LIN {X 0,Y 386.045,Z 430.319,A -85,B 0,C 180,E1 -12861.883,E2 -12861.883} C_VEL
LIN {X 0,Y 387.779,Z 432.947,A -85,B 0,C 180,E1 -12862.928,E2 -12862.928} C_VEL
LIN {X 0,Y 389.811,Z 435.003,A -85,B 0,C 180,E1 -12864.309,E2 -12864.309} C_VEL
LIN {X 0,Y 391.644,Z 436.137,A -85,B 0,C 180,E1 -12865.884,E2 -12865.884} C_VEL
LIN {X 0,Y 393.22,Z 436.525,A -85,B 0,C 180,E1 -12867.952,E2 -12867.952} C_VEL
LIN {X 0,Y 393.637,Z 436.553,A -85,B 0,C 180,E1 -12868.977,E2 -12868.977} C_VEL
LIN {X 0,Y 393.779,Z 436.58,A -85,B 0,C 180,E1 -12870,E2 -12870} C_VEL
LIN {X 0,Y 393.63,Z 436.554,A -85,B 0,C 180,E1 -12871.061,E2 -12871.061} C_VEL
LIN {X 0,Y 392.568,Z 436.348,A -85,B 0,C 180,E1 -12873.079,E2 -12873.079} C_VEL
LIN {X 0,Y 391.09,Z 435.883,A -85,B 0,C 180,E1 -12874.638,E2 -12874.638} C_VEL
LIN {X 0,Y 389.048,Z 434.381,A -85,B 0,C 180,E1 -12876.222,E2 -12876.222} C_VEL
LIN {X 0,Y 386.851,Z 431.737,A -85,B 0,C 180,E1 -12877.626,E2 -12877.626} C_VEL
LIN {X 0,Y 385.902,Z 430.065,A -85,B 0,C 180,E1 -12878.206,E2 -12878.206} C_VEL
LIN {X 0,Y 383.077,Z 428.613,A -85,B 0,C 180,E1 -12879.504,E2 -12879.504} C_VEL
LIN {X 0,Y 380.566,Z 426.106,A -85,B 0,C 180,E1 -12880.574,E2 -12880.574} C_VEL
LIN {X 0,Y 379.095,Z 423.761,A -85,B 0,C 180,E1 -12881.204,E2 -12881.204} C_VEL
LIN {X 0,Y 376.337,Z 421.957,A -85,B 0,C 180,E1 -12882.162,E2 -12882.162} C_VEL
LIN {X 0,Y 374.318,Z 419.242,A -85,B 0,C 180,E1 -12882.888,E2 -12882.888} C_VEL
LIN {X 0,Y 373.606,Z 417.793,A -85,B 0,C 180,E1 -12883.139,E2 -12883.139} C_VEL
LIN {X 0,Y 370.881,Z 415.993,A -85,B 0,C 180,E1 -12883.966,E2 -12883.966} C_VEL
LIN {X 0,Y 369.4,Z 413.626,A -85,B 0,C 180,E1 -12884.425,E2 -12884.425} C_VEL
LIN {X 0,Y 369.015,Z 412.02,A -85,B 0,C 180,E1 -12884.616,E2 -12884.616} C_VEL
LIN {X 0,Y 368.997,Z 412.024,A -85,B 0,C 180,E1 -12887.768,E2 -12887.768} C_VEL
LIN {X 0,Y 368.925,Z 412.029,A -85,B 0,C 180,E1 -12891.219,E2 -12891.219} C_VEL
LIN {X 0,Y 368.953,Z 412.023,A -85,B 0,C 180,E1 -12894.775,E2 -12894.775} C_VEL
LIN {X 0,Y 368.958,Z 412.025,A -85,B 0,C 180,E1 -12897.203,E2 -12897.203} C_VEL
LIN {X 0,Y 368.923,Z 412.028,A -85,B 0,C 180,E1 -12900.953,E2 -12900.953} C_VEL
LIN {X 0,Y 368.923,Z 412.029,A -85,B 0,C 180,E1 -12905.001,E2 -12905.001} C_VEL
LIN {X 0,Y 368.904,Z 412.03,A -85,B 0,C 180,E1 -12908.64,E2 -12908.64} C_VEL
LIN {X 0,Y 368.875,Z 412.033,A -85,B 0,C 180,E1 -12912.009,E2 -12912.009} C_VEL
LIN {X 0,Y 368.897,Z 412.032,A -85,B 0,C 180,E1 -12914.773,E2 -12914.773} C_VEL
LIN {X 0,Y 368.28,Z 412.114,A -85,B 0,C 180,E1 -12915.684,E2 -12915.684} C_VEL
LIN {X 0,Y 365.413,Z 412.476,A -85,B 0,C 180,E1 -12917.165,E2 -12917.165} C_VEL
LIN {X 0,Y 362.955,Z 412.78,A -85,B 0,C 180,E1 -12918.362,E2 -12918.362} C_VEL
LIN {X 0,Y 361.906,Z 412.906,A -85,B 0,C 180,E1 -12919.29,E2 -12919.29} C_VEL
LIN {X 0,Y 361.826,Z 412.913,A -85,B 0,C 180,E1 -12919.604,E2 -12919.604} C_VEL
LIN {X 0,Y 361.86,Z 412.911,A -85,B 0,C 180,E1 -12922.982,E2 -12922.982} C_VEL
LIN {X 0,Y 361.851,Z 412.91,A -85,B 0,C 180,E1 -12926.631,E2 -12926.631} C_VEL
LIN {X 0,Y 361.868,Z 412.906,A -85,B 0,C 180,E1 -12929.672,E2 -12929.672} C_VEL
LIN {X 0,Y 361.946,Z 412.897,A -85,B 0,C 180,E1 -12933.475,E2 -12933.475} C_VEL
LIN {X 0,Y 361.882,Z 412.908,A -85,B 0,C 180,E1 -12937.145,E2 -12937.145} C_VEL
LIN {X 0,Y 361.898,Z 412.907,A -85,B 0,C 180,E1 -12940.724,E2 -12940.724} C_VEL
LIN {X 0,Y 361.924,Z 412.902,A -85,B 0,C 180,E1 -12943.066,E2 -12943.066} C_VEL
LIN {X 0,Y 361.99,Z 412.894,A -85,B 0,C 180,E1 -12946.528,E2 -12946.528} C_VEL
LIN {X 0,Y 362.023,Z 412.887,A -85,B 0,C 180,E1 -12949.938,E2 -12949.938} C_VEL
LIN {X 0,Y 362.155,Z 412.87,A -85,B 0,C 180,E1 -12953.314,E2 -12953.314} C_VEL
LIN {X 0,Y 362.275,Z 412.855,A -85,B 0,C 180,E1 -12957.777,E2 -12957.777} C_VEL
LIN {X 0,Y 362.42,Z 412.838,A -85,B 0,C 180,E1 -12960.001,E2 -12960.001} C_VEL
LIN {X 0,Y 362.275,Z 412.858,A -85,B 0,C 180,E1 -12962.224,E2 -12962.224} C_VEL
LIN {X 0,Y 362.155,Z 412.873,A -85,B 0,C 180,E1 -12966.687,E2 -12966.687} C_VEL
LIN {X 0,Y 362.024,Z 412.889,A -85,B 0,C 180,E1 -12970.063,E2 -12970.063} C_VEL
LIN {X 0,Y 361.991,Z 412.893,A -85,B 0,C 180,E1 -12973.899,E2 -12973.899} C_VEL
LIN {X 0,Y 361.962,Z 412.897,A -85,B 0,C 180,E1 -12977.939,E2 -12977.939} C_VEL
LIN {X 0,Y 361.856,Z 412.909,A -85,B 0,C 180,E1 -12981.656,E2 -12981.656} C_VEL
LIN {X 0,Y 361.922,Z 412.899,A -85,B 0,C 180,E1 -12985.291,E2 -12985.291} C_VEL
LIN {X 0,Y 361.918,Z 412.903,A -85,B 0,C 180,E1 -12987.779,E2 -12987.779} C_VEL
LIN {X 0,Y 361.856,Z 412.91,A -85,B 0,C 180,E1 -12991.628,E2 -12991.628} C_VEL
LIN {X 0,Y 361.871,Z 412.908,A -85,B 0,C 180,E1 -12995.346,E2 -12995.346} C_VEL
LIN {X 0,Y 361.904,Z 413.183,A -85,B 0,C 180,E1 -12997.233,E2 -12997.233} C_VEL
LIN {X 0,Y 362.344,Z 416.07,A -85,B 0,C 180,E1 -13000.85,E2 -13000.85} C_VEL
LIN {X 0,Y 362.736,Z 418.994,A -85,B 0,C 180,E1 -13004.227,E2 -13004.227} C_VEL
LIN {X 0,Y 362.941,Z 422.013,A -85,B 0,C 180,E1 -13007.378,E2 -13007.378} C_VEL
LIN {X 0,Y 362.693,Z 425.597,A -85,B 0,C 180,E1 -13010.814,E2 -13010.814} C_VEL
LIN {X 0,Y 362.451,Z 428.076,A -85,B 0,C 180,E1 -13013.053,E2 -13013.053} C_VEL
LIN {X 0,Y 361.94,Z 432.762,A -85,B 0,C 180,E1 -13017.065,E2 -13017.065} C_VEL
LIN {X 0,Y 361.583,Z 435.917,A -85,B 0,C 180,E1 -13019.646,E2 -13019.646} C_VEL
LIN {X 0,Y 361.173,Z 440.843,A -85,B 0,C 180,E1 -13023.523,E2 -13023.523} C_VEL
LIN {X 0,Y 360.817,Z 445.545,A -85,B 0,C 180,E1 -13027.073,E2 -13027.073} C_VEL
LIN {X 0,Y 360.66,Z 449.44,A -85,B 0,C 180,E1 -13029.95,E2 -13029.95} C_VEL
LIN {X 0,Y 362.752,Z 459.144,A -85,B 0,C 180,E1 -13030.411,E2 -13030.411} C_VEL
LIN {X 0,Y 364.561,Z 469.064,A -85,B 0,C 180,E1 -13030.996,E2 -13030.996} C_VEL
LIN {X 0,Y 366.022,Z 478.867,A -85,B 0,C 180,E1 -13031.698,E2 -13031.698} C_VEL
LIN {X 0,Y 366.573,Z 486.079,A -85,B 0,C 180,E1 -13032.281,E2 -13032.281} C_VEL
LIN {X 0,Y 365.702,Z 495.355,A -85,B 0,C 180,E1 -13033.102,E2 -13033.102} C_VEL
LIN {X 0,Y 364.823,Z 504.301,A -85,B 0,C 180,E1 -13034.067,E2 -13034.067} C_VEL
LIN {X 0,Y 364.052,Z 511.792,A -85,B 0,C 180,E1 -13035.025,E2 -13035.025} C_VEL
LIN {X 0,Y 363.189,Z 520.053,A -85,B 0,C 180,E1 -13036.288,E2 -13036.288} C_VEL
LIN {X 0,Y 362.493,Z 526.255,A -85,B 0,C 180,E1 -13037.402,E2 -13037.402} C_VEL
LIN {X 0,Y 361.716,Z 532.791,A -85,B 0,C 180,E1 -13038.797,E2 -13038.797} C_VEL
LIN {X 0,Y 361.284,Z 537.294,A -85,B 0,C 180,E1 -13039.917,E2 -13039.917} C_VEL
LIN {X 0,Y 360.824,Z 542.787,A -85,B 0,C 180,E1 -13041.6,E2 -13041.6} C_VEL
LIN {X 0,Y 360.5,Z 547.112,A -85,B 0,C 180,E1 -13043.283,E2 -13043.283} C_VEL
LIN {X 0,Y 360.385,Z 549.479,A -85,B 0,C 180,E1 -13044.405,E2 -13044.405} C_VEL
LIN {X 0,Y 360.369,Z 551.28,A -85,B 0,C 180,E1 -13045.526,E2 -13045.526} C_VEL
LIN {X 0,Y 360.265,Z 553.724,A -85,B 0,C 180,E1 -13047.764,E2 -13047.764} C_VEL
LIN {X 0,Y 360.304,Z 554.314,A -85,B 0,C 180,E1 -13048.882,E2 -13048.882} C_VEL
LIN {X 0,Y 360.304,Z 554.314,A -85,B 0,C 180,E1 -13051.118,E2 -13051.118} C_VEL
LIN {X 0,Y 360.265,Z 553.724,A -85,B 0,C 180,E1 -13052.236,E2 -13052.236} C_VEL
LIN {X 0,Y 360.369,Z 551.28,A -85,B 0,C 180,E1 -13054.474,E2 -13054.474} C_VEL
LIN {X 0,Y 360.381,Z 548.748,A -85,B 0,C 180,E1 -13055.963,E2 -13055.963} C_VEL
LIN {X 0,Y 360.597,Z 545.872,A -85,B 0,C 180,E1 -13057.278,E2 -13057.278} C_VEL
LIN {X 0,Y 360.964,Z 541.127,A -85,B 0,C 180,E1 -13058.961,E2 -13058.961} C_VEL
LIN {X 0,Y 361.523,Z 535.104,A -85,B 0,C 180,E1 -13060.642,E2 -13060.642} C_VEL
LIN {X 0,Y 362.127,Z 529.006,A -85,B 0,C 180,E1 -13062.042,E2 -13062.042} C_VEL
LIN {X 0,Y 362.825,Z 523.307,A -85,B 0,C 180,E1 -13063.156,E2 -13063.156} C_VEL
LIN {X 0,Y 363.714,Z 514.751,A -85,B 0,C 180,E1 -13064.548,E2 -13064.548} C_VEL
LIN {X 0,Y 364.499,Z 506.568,A -85,B 0,C 180,E1 -13065.66,E2 -13065.66} C_VEL
LIN {X 0,Y 365.4,Z 498.058,A -85,B 0,C 180,E1 -13066.624,E2 -13066.624} C_VEL
LIN {X 0,Y 366.31,Z 489.344,A -85,B 0,C 180,E1 -13067.444,E2 -13067.444} C_VEL
LIN {X 0,Y 366.462,Z 483.435,A -85,B 0,C 180,E1 -13067.951,E2 -13067.951} C_VEL
LIN {X 0,Y 364.941,Z 471.284,A -85,B 0,C 180,E1 -13068.858,E2 -13068.858} C_VEL
LIN {X 0,Y 363.012,Z 460.41,A -85,B 0,C 180,E1 -13069.522,E2 -13069.522} C_VEL
LIN {X 0,Y 360.702,Z 449.94,A -85,B 0,C 180,E1 -13070.033,E2 -13070.033} C_VEL
LIN {X 0,Y 360.657,Z 449.333,A -85,B 0,C 180,E1 -13070.087,E2 -13070.087} C_VEL
LIN {X 0,Y 360.921,Z 443.914,A -85,B 0,C 180,E1 -13074.136,E2 -13074.136} C_VEL
LIN {X 0,Y 361.303,Z 439.09,A -85,B 0,C 180,E1 -13077.829,E2 -13077.829} C_VEL
LIN {X 0,Y 361.765,Z 434.324,A -85,B 0,C 180,E1 -13081.636,E2 -13081.636} C_VEL
LIN {X 0,Y 362.097,Z 431.184,A -85,B 0,C 180,E1 -13084.253,E2 -13084.253} C_VEL
LIN {X 0,Y 362.502,Z 427.609,A -85,B 0,C 180,E1 -13087.355,E2 -13087.355} C_VEL
LIN {X 0,Y 362.736,Z 424.992,A -85,B 0,C 180,E1 -13089.744,E2 -13089.744} C_VEL
LIN {X 0,Y 362.943,Z 421.946,A -85,B 0,C 180,E1 -13092.666,E2 -13092.666} C_VEL
LIN {X 0,Y 362.732,Z 418.972,A -85,B 0,C 180,E1 -13095.796,E2 -13095.796} C_VEL
LIN {X 0,Y 362.344,Z 416.069,A -85,B 0,C 180,E1 -13099.15,E2 -13099.15} C_VEL
LIN {X 0,Y 361.877,Z 413.027,A -85,B 0,C 180,E1 -13102.982,E2 -13102.982} C_VEL
LIN {X 0,Y 361.86,Z 412.908,A -85,B 0,C 180,E1 -13106.628,E2 -13106.628} C_VEL
LIN {X 0,Y 361.872,Z 412.908,A -85,B 0,C 180,E1 -13109.671,E2 -13109.671} C_VEL
LIN {X 0,Y 361.95,Z 412.898,A -85,B 0,C 180,E1 -13113.474,E2 -13113.474} C_VEL
LIN {X 0,Y 361.877,Z 412.905,A -85,B 0,C 180,E1 -13117.143,E2 -13117.143} C_VEL
LIN {X 0,Y 361.904,Z 412.901,A -85,B 0,C 180,E1 -13120.723,E2 -13120.723} C_VEL
LIN {X 0,Y 361.929,Z 412.899,A -85,B 0,C 180,E1 -13123.065,E2 -13123.065} C_VEL
LIN {X 0,Y 361.992,Z 412.89,A -85,B 0,C 180,E1 -13126.527,E2 -13126.527} C_VEL
LIN {X 0,Y 362.024,Z 412.889,A -85,B 0,C 180,E1 -13129.937,E2 -13129.937} C_VEL
LIN {X 0,Y 362.155,Z 412.873,A -85,B 0,C 180,E1 -13133.313,E2 -13133.313} C_VEL
LIN {X 0,Y 362.275,Z 412.858,A -85,B 0,C 180,E1 -13137.776,E2 -13137.776} C_VEL
LIN {X 0,Y 362.42,Z 412.838,A -85,B 0,C 180,E1 -13139.999,E2 -13139.999} C_VEL
LIN {X 0,Y 362.275,Z 412.855,A -85,B 0,C 180,E1 -13142.223,E2 -13142.223} C_VEL
LIN {X 0,Y 362.155,Z 412.87,A -85,B 0,C 180,E1 -13146.686,E2 -13146.686} C_VEL
LIN {X 0,Y 362.023,Z 412.887,A -85,B 0,C 180,E1 -13150.062,E2 -13150.062} C_VEL
LIN {X 0,Y 361.99,Z 412.891,A -85,B 0,C 180,E1 -13153.898,E2 -13153.898} C_VEL
LIN {X 0,Y 361.959,Z 412.895,A -85,B 0,C 180,E1 -13157.938,E2 -13157.938} C_VEL
LIN {X 0,Y 361.884,Z 412.905,A -85,B 0,C 180,E1 -13161.653,E2 -13161.653} C_VEL
LIN {X 0,Y 361.92,Z 412.903,A -85,B 0,C 180,E1 -13165.29,E2 -13165.29} C_VEL
LIN {X 0,Y 361.914,Z 412.9,A -85,B 0,C 180,E1 -13167.778,E2 -13167.778} C_VEL
LIN {X 0,Y 361.839,Z 412.912,A -85,B 0,C 180,E1 -13171.285,E2 -13171.285} C_VEL
LIN {X 0,Y 361.846,Z 412.909,A -85,B 0,C 180,E1 -13174.28,E2 -13174.28} C_VEL
LIN {X 0,Y 361.858,Z 412.909,A -85,B 0,C 180,E1 -13177.223,E2 -13177.223} C_VEL
LIN {X 0,Y 361.898,Z 412.908,A -85,B 0,C 180,E1 -13180.768,E2 -13180.768} C_VEL
LIN {X 0,Y 361.897,Z 412.904,A -85,B 0,C 180,E1 -13184.355,E2 -13184.355} C_VEL
LIN {X 0,Y 361.831,Z 412.91,A -85,B 0,C 180,E1 -13187.568,E2 -13187.568} C_VEL
LIN {X 0,Y 361.865,Z 412.909,A -85,B 0,C 180,E1 -13190.973,E2 -13190.973} C_VEL
LIN {X 0,Y 361.868,Z 412.911,A -85,B 0,C 180,E1 -13194.655,E2 -13194.655} C_VEL
LIN {X 0,Y 361.832,Z 412.915,A -85,B 0,C 180,E1 -13198.371,E2 -13198.371} C_VEL
LIN {X 0,Y 361.903,Z 412.905,A -85,B 0,C 180,E1 -13202.221,E2 -13202.221} C_VEL
LIN {X 0,Y 361.923,Z 412.902,A -85,B 0,C 180,E1 -13204.71,E2 -13204.71} C_VEL
LIN {X 0,Y 361.887,Z 412.91,A -85,B 0,C 180,E1 -13208.347,E2 -13208.347} C_VEL
LIN {X 0,Y 361.963,Z 412.9,A -85,B 0,C 180,E1 -13212.062,E2 -13212.062} C_VEL
LIN {X 0,Y 361.968,Z 413.088,A -85,B 0,C 180,E1 -13213.793,E2 -13213.793} C_VEL
LIN {X 0,Y 362.869,Z 415.66,A -85,B 0,C 180,E1 -13214.083,E2 -13214.083} C_VEL
LIN {X 0,Y 364.91,Z 417.806,A -85,B 0,C 180,E1 -13214.616,E2 -13214.616} C_VEL
LIN {X 0,Y 366.344,Z 418.896,A -85,B 0,C 180,E1 -13215.001,E2 -13215.001} C_VEL
LIN {X 0,Y 368.15,Z 421.839,A -85,B 0,C 180,E1 -13215.56,E2 -13215.56} C_VEL
LIN {X 0,Y 370.818,Z 424.02,A -85,B 0,C 180,E1 -13216.326,E2 -13216.326} C_VEL
LIN {X 0,Y 371.761,Z 425.081,A -85,B 0,C 180,E1 -13216.631,E2 -13216.631} C_VEL
LIN {X 0,Y 374.12,Z 428.158,A -85,B 0,C 180,E1 -13217.417,E2 -13217.417} C_VEL
LIN {X 0,Y 377.044,Z 430.332,A -85,B 0,C 180,E1 -13218.416,E2 -13218.416} C_VEL
LIN {X 0,Y 380.045,Z 434.031,A -85,B 0,C 180,E1 -13219.613,E2 -13219.613} C_VEL
LIN {X 0,Y 382.714,Z 436.121,A -85,B 0,C 180,E1 -13220.746,E2 -13220.746} C_VEL
LIN {X 0,Y 384.738,Z 437.322,A -85,B 0,C 180,E1 -13221.683,E2 -13221.683} C_VEL
LIN {X 0,Y 386.981,Z 440.32,A -85,B 0,C 180,E1 -13223.007,E2 -13223.007} C_VEL
LIN {X 0,Y 388.899,Z 442.057,A -85,B 0,C 180,E1 -13224.296,E2 -13224.296} C_VEL
LIN {X 0,Y 390.755,Z 443.18,A -85,B 0,C 180,E1 -13225.875,E2 -13225.875} C_VEL
LIN {X 0,Y 392.358,Z 443.566,A -85,B 0,C 180,E1 -13227.947,E2 -13227.947} C_VEL
LIN {X 0,Y 392.776,Z 443.6,A -85,B 0,C 180,E1 -13228.975,E2 -13228.975} C_VEL
LIN {X 0,Y 392.914,Z 443.626,A -85,B 0,C 180,E1 -13230,E2 -13230} C_VEL
LIN {X 0,Y 392.776,Z 443.603,A -85,B 0,C 180,E1 -13231.025,E2 -13231.025} C_VEL
LIN {X 0,Y 391.691,Z 443.392,A -85,B 0,C 180,E1 -13233.086,E2 -13233.086} C_VEL
LIN {X 0,Y 390.205,Z 442.909,A -85,B 0,C 180,E1 -13234.649,E2 -13234.649} C_VEL
LIN {X 0,Y 387.984,Z 441.374,A -85,B 0,C 180,E1 -13236.337,E2 -13236.337} C_VEL
LIN {X 0,Y 385.591,Z 438.638,A -85,B 0,C 180,E1 -13237.815,E2 -13237.815} C_VEL
LIN {X 0,Y 384.275,Z 436.859,A -85,B 0,C 180,E1 -13238.545,E2 -13238.545} C_VEL
LIN {X 0,Y 381.278,Z 435.114,A -85,B 0,C 180,E1 -13239.884,E2 -13239.884} C_VEL
LIN {X 0,Y 378.546,Z 432.311,A -85,B 0,C 180,E1 -13240.999,E2 -13240.999} C_VEL
LIN {X 0,Y 377.317,Z 430.475,A -85,B 0,C 180,E1 -13241.493,E2 -13241.493} C_VEL
LIN {X 0,Y 374.247,Z 428.264,A -85,B 0,C 180,E1 -13242.541,E2 -13242.541} C_VEL
LIN {X 0,Y 371.914,Z 425.332,A -85,B 0,C 180,E1 -13243.316,E2 -13243.316} C_VEL
LIN {X 0,Y 371.043,Z 424.16,A -85,B 0,C 180,E1 -13243.605,E2 -13243.605} C_VEL
LIN {X 0,Y 368.278,Z 421.965,A -85,B 0,C 180,E1 -13244.403,E2 -13244.403} C_VEL
LIN {X 0,Y 366.452,Z 419.106,A -85,B 0,C 180,E1 -13244.964,E2 -13244.964} C_VEL
LIN {X 0,Y 365.576,Z 418.223,A -85,B 0,C 180,E1 -13245.216,E2 -13245.216} C_VEL
LIN {X 0,Y 363.298,Z 416.292,A -85,B 0,C 180,E1 -13245.8,E2 -13245.8} C_VEL
LIN {X 0,Y 362.122,Z 413.871,A -85,B 0,C 180,E1 -13246.145,E2 -13246.145} C_VEL
LIN {X 0,Y 361.931,Z 412.904,A -85,B 0,C 180,E1 -13246.244,E2 -13246.244} C_VEL
LIN {X 0,Y 361.916,Z 412.905,A -85,B 0,C 180,E1 -13249.276,E2 -13249.276} C_VEL
LIN {X 0,Y 361.887,Z 412.904,A -85,B 0,C 180,E1 -13252.855,E2 -13252.855} C_VEL
LIN {X 0,Y 361.936,Z 412.897,A -85,B 0,C 180,E1 -13256.721,E2 -13256.721} C_VEL
LIN {X 0,Y 361.867,Z 412.906,A -85,B 0,C 180,E1 -13260.328,E2 -13260.328} C_VEL
LIN {X 0,Y 361.848,Z 412.908,A -85,B 0,C 180,E1 -13264.28,E2 -13264.28} C_VEL
LIN {X 0,Y 361.865,Z 412.91,A -85,B 0,C 180,E1 -13267.224,E2 -13267.224} C_VEL
LIN {X 0,Y 361.83,Z 412.911,A -85,B 0,C 180,E1 -13270.755,E2 -13270.755} C_VEL
LIN {X 0,Y 361.828,Z 412.911,A -85,B 0,C 180,E1 -13274.365,E2 -13274.365} C_VEL
LIN {X 0,Y 361.829,Z 412.913,A -85,B 0,C 180,E1 -13277.568,E2 -13277.568} C_VEL
LIN {X 0,Y 361.826,Z 412.913,A -85,B 0,C 180,E1 -13279.604,E2 -13279.604} C_VEL
LIN {X 0,Y 361.178,Z 412.994,A -85,B 0,C 180,E1 -13280.533,E2 -13280.533} C_VEL
LIN {X 0,Y 358.347,Z 413.344,A -85,B 0,C 180,E1 -13282.044,E2 -13282.044} C_VEL
LIN {X 0,Y 355.936,Z 413.649,A -85,B 0,C 180,E1 -13283.266,E2 -13283.266} C_VEL
LIN {X 0,Y 354.894,Z 413.775,A -85,B 0,C 180,E1 -13284.211,E2 -13284.211} C_VEL
LIN {X 0,Y 354.806,Z 413.786,A -85,B 0,C 180,E1 -13284.532,E2 -13284.532} C_VEL
LIN {X 0,Y 354.779,Z 413.79,A -85,B 0,C 180,E1 -13287.667,E2 -13287.667} C_VEL
LIN {X 0,Y 354.861,Z 413.781,A -85,B 0,C 180,E1 -13290.621,E2 -13290.621} C_VEL
LIN {X 0,Y 354.891,Z 413.775,A -85,B 0,C 180,E1 -13294.173,E2 -13294.173} C_VEL
LIN {X 0,Y 354.826,Z 413.783,A -85,B 0,C 180,E1 -13297.894,E2 -13297.894} C_VEL
LIN {X 0,Y 354.914,Z 413.772,A -85,B 0,C 180,E1 -13301.892,E2 -13301.892} C_VEL
LIN {X 0,Y 354.934,Z 413.77,A -85,B 0,C 180,E1 -13305.982,E2 -13305.982} C_VEL
LIN {X 0,Y 354.97,Z 413.765,A -85,B 0,C 180,E1 -13309.736,E2 -13309.736} C_VEL
LIN {X 0,Y 355.119,Z 413.748,A -85,B 0,C 180,E1 -13313.181,E2 -13313.181} C_VEL
LIN {X 0,Y 355.238,Z 413.731,A -85,B 0,C 180,E1 -13317.733,E2 -13317.733} C_VEL
LIN {X 0,Y 355.39,Z 413.714,A -85,B 0,C 180,E1 -13320.001,E2 -13320.001} C_VEL
LIN {X 0,Y 355.238,Z 413.735,A -85,B 0,C 180,E1 -13322.268,E2 -13322.268} C_VEL
LIN {X 0,Y 355.119,Z 413.749,A -85,B 0,C 180,E1 -13326.82,E2 -13326.82} C_VEL
LIN {X 0,Y 354.971,Z 413.77,A -85,B 0,C 180,E1 -13330.265,E2 -13330.265} C_VEL
LIN {X 0,Y 354.937,Z 413.772,A -85,B 0,C 180,E1 -13334.02,E2 -13334.02} C_VEL
LIN {X 0,Y 354.917,Z 413.777,A -85,B 0,C 180,E1 -13338.109,E2 -13338.109} C_VEL
LIN {X 0,Y 354.811,Z 413.79,A -85,B 0,C 180,E1 -13342.108,E2 -13342.108} C_VEL
LIN {X 0,Y 354.894,Z 413.778,A -85,B 0,C 180,E1 -13345.828,E2 -13345.828} C_VEL
LIN {X 0,Y 354.85,Z 413.783,A -85,B 0,C 180,E1 -13349.679,E2 -13349.679} C_VEL
LIN {X 0,Y 354.827,Z 413.786,A -85,B 0,C 180,E1 -13353.683,E2 -13353.683} C_VEL
LIN {X 0,Y 354.797,Z 413.793,A -85,B 0,C 180,E1 -13356.46,E2 -13356.46} C_VEL
LIN {X 0,Y 355.157,Z 416.084,A -85,B 0,C 180,E1 -13359.49,E2 -13359.49} C_VEL
LIN {X 0,Y 355.563,Z 418.956,A -85,B 0,C 180,E1 -13363.003,E2 -13363.003} C_VEL
LIN {X 0,Y 355.839,Z 421.93,A -85,B 0,C 180,E1 -13366.271,E2 -13366.271} C_VEL
LIN {X 0,Y 355.767,Z 424.947,A -85,B 0,C 180,E1 -13369.316,E2 -13369.316} C_VEL
LIN {X 0,Y 355.48,Z 428.068,A -85,B 0,C 180,E1 -13372.263,E2 -13372.263} C_VEL
LIN {X 0,Y 355.141,Z 431.1,A -85,B 0,C 180,E1 -13374.979,E2 -13374.979} C_VEL
LIN {X 0,Y 354.632,Z 435.807,A -85,B 0,C 180,E1 -13378.986,E2 -13378.986} C_VEL
LIN {X 0,Y 354.142,Z 440.582,A -85,B 0,C 180,E1 -13382.843,E2 -13382.843} C_VEL
LIN {X 0,Y 353.785,Z 445.375,A -85,B 0,C 180,E1 -13386.591,E2 -13386.591} C_VEL
LIN {X 0,Y 353.629,Z 449.234,A -85,B 0,C 180,E1 -13389.534,E2 -13389.534} C_VEL
LIN {X 0,Y 355.859,Z 459.618,A -85,B 0,C 180,E1 -13390.045,E2 -13390.045} C_VEL
LIN {X 0,Y 357.761,Z 470.036,A -85,B 0,C 180,E1 -13390.689,E2 -13390.689} C_VEL
LIN {X 0,Y 359.236,Z 480.219,A -85,B 0,C 180,E1 -13391.453,E2 -13391.453} C_VEL
LIN {X 0,Y 359.659,Z 487.514,A -85,B 0,C 180,E1 -13392.076,E2 -13392.076} C_VEL
LIN {X 0,Y 358.765,Z 496.51,A -85,B 0,C 180,E1 -13392.912,E2 -13392.912} C_VEL
LIN {X 0,Y 357.84,Z 505.238,A -85,B 0,C 180,E1 -13393.894,E2 -13393.894} C_VEL
LIN {X 0,Y 357.09,Z 512.332,A -85,B 0,C 180,E1 -13394.838,E2 -13394.838} C_VEL
LIN {X 0,Y 356.244,Z 519.854,A -85,B 0,C 180,E1 -13396.015,E2 -13396.015} C_VEL
LIN {X 0,Y 355.527,Z 526.057,A -85,B 0,C 180,E1 -13397.151,E2 -13397.151} C_VEL
LIN {X 0,Y 354.715,Z 532.593,A -85,B 0,C 180,E1 -13398.573,E2 -13398.573} C_VEL
LIN {X 0,Y 354.27,Z 537.096,A -85,B 0,C 180,E1 -13399.715,E2 -13399.715} C_VEL
LIN {X 0,Y 353.783,Z 542.59,A -85,B 0,C 180,E1 -13401.432,E2 -13401.432} C_VEL
LIN {X 0,Y 353.419,Z 546.914,A -85,B 0,C 180,E1 -13403.148,E2 -13403.148} C_VEL
LIN {X 0,Y 353.283,Z 549.281,A -85,B 0,C 180,E1 -13404.292,E2 -13404.292} C_VEL
LIN {X 0,Y 353.281,Z 551.083,A -85,B 0,C 180,E1 -13405.436,E2 -13405.436} C_VEL
LIN {X 0,Y 353.174,Z 553.527,A -85,B 0,C 180,E1 -13407.719,E2 -13407.719} C_VEL
LIN {X 0,Y 353.204,Z 554.117,A -85,B 0,C 180,E1 -13408.86,E2 -13408.86} C_VEL
LIN {X 0,Y 353.262,Z 554.272,A -85,B 0,C 180,E1 -13410,E2 -13410} C_VEL
LIN {X 0,Y 353.204,Z 554.117,A -85,B 0,C 180,E1 -13411.14,E2 -13411.14} C_VEL
LIN {X 0,Y 353.174,Z 553.527,A -85,B 0,C 180,E1 -13412.281,E2 -13412.281} C_VEL
LIN {X 0,Y 353.282,Z 551.083,A -85,B 0,C 180,E1 -13414.564,E2 -13414.564} C_VEL
LIN {X 0,Y 353.298,Z 548.86,A -85,B 0,C 180,E1 -13415.937,E2 -13415.937} C_VEL
LIN {X 0,Y 353.521,Z 545.674,A -85,B 0,C 180,E1 -13417.424,E2 -13417.424} C_VEL
LIN {X 0,Y 353.918,Z 540.929,A -85,B 0,C 180,E1 -13419.141,E2 -13419.141} C_VEL
LIN {X 0,Y 354.494,Z 534.905,A -85,B 0,C 180,E1 -13420.856,E2 -13420.856} C_VEL
LIN {X 0,Y 355.162,Z 528.808,A -85,B 0,C 180,E1 -13422.282,E2 -13422.282} C_VEL
LIN {X 0,Y 355.89,Z 523.109,A -85,B 0,C 180,E1 -13423.417,E2 -13423.417} C_VEL
LIN {X 0,Y 356.823,Z 514.554,A -85,B 0,C 180,E1 -13424.835,E2 -13424.835} C_VEL
LIN {X 0,Y 357.658,Z 506.371,A -85,B 0,C 180,E1 -13425.968,E2 -13425.968} C_VEL
LIN {X 0,Y 358.594,Z 497.861,A -85,B 0,C 180,E1 -13426.949,E2 -13426.949} C_VEL
LIN {X 0,Y 359.527,Z 489.147,A -85,B 0,C 180,E1 -13427.784,E2 -13427.784} C_VEL
LIN {X 0,Y 359.613,Z 484.238,A -85,B 0,C 180,E1 -13428.221,E2 -13428.221} C_VEL
LIN {X 0,Y 358.176,Z 472.574,A -85,B 0,C 180,E1 -13429.143,E2 -13429.143} C_VEL
LIN {X 0,Y 356.111,Z 460.945,A -85,B 0,C 180,E1 -13429.884,E2 -13429.884} C_VEL
LIN {X 0,Y 353.684,Z 449.872,A -85,B 0,C 180,E1 -13430.444,E2 -13430.444} C_VEL
LIN {X 0,Y 353.633,Z 449.164,A -85,B 0,C 180,E1 -13430.504,E2 -13430.504} C_VEL
LIN {X 0,Y 353.892,Z 443.761,A -85,B 0,C 180,E1 -13434.647,E2 -13434.647} C_VEL
LIN {X 0,Y 354.279,Z 438.968,A -85,B 0,C 180,E1 -13438.43,E2 -13438.43} C_VEL
LIN {X 0,Y 354.696,Z 435.129,A -85,B 0,C 180,E1 -13441.568,E2 -13441.568} C_VEL
LIN {X 0,Y 355.115,Z 431.099,A -85,B 0,C 180,E1 -13445.024,E2 -13445.024} C_VEL
LIN {X 0,Y 355.485,Z 427.997,A -85,B 0,C 180,E1 -13447.797,E2 -13447.797} C_VEL
LIN {X 0,Y 355.832,Z 424.242,A -85,B 0,C 180,E1 -13451.363,E2 -13451.363} C_VEL
LIN {X 0,Y 355.84,Z 421.918,A -85,B 0,C 180,E1 -13453.729,E2 -13453.729} C_VEL
LIN {X 0,Y 355.545,Z 418.949,A -85,B 0,C 180,E1 -13457,E2 -13457} C_VEL
LIN {X 0,Y 355.157,Z 416.085,A -85,B 0,C 180,E1 -13460.509,E2 -13460.509} C_VEL
LIN {X 0,Y 354.797,Z 413.792,A -85,B 0,C 180,E1 -13463.54,E2 -13463.54} C_VEL
LIN {X 0,Y 354.827,Z 413.786,A -85,B 0,C 180,E1 -13466.317,E2 -13466.317} C_VEL
LIN {X 0,Y 354.85,Z 413.783,A -85,B 0,C 180,E1 -13470.321,E2 -13470.321} C_VEL
LIN {X 0,Y 354.894,Z 413.778,A -85,B 0,C 180,E1 -13474.172,E2 -13474.172} C_VEL
LIN {X 0,Y 354.811,Z 413.79,A -85,B 0,C 180,E1 -13477.892,E2 -13477.892} C_VEL
LIN {X 0,Y 354.917,Z 413.776,A -85,B 0,C 180,E1 -13481.891,E2 -13481.891} C_VEL
LIN {X 0,Y 354.937,Z 413.772,A -85,B 0,C 180,E1 -13485.98,E2 -13485.98} C_VEL
LIN {X 0,Y 354.971,Z 413.77,A -85,B 0,C 180,E1 -13489.735,E2 -13489.735} C_VEL
LIN {X 0,Y 355.119,Z 413.749,A -85,B 0,C 180,E1 -13493.18,E2 -13493.18} C_VEL
LIN {X 0,Y 355.238,Z 413.735,A -85,B 0,C 180,E1 -13497.732,E2 -13497.732} C_VEL
LIN {X 0,Y 355.39,Z 413.714,A -85,B 0,C 180,E1 -13499.999,E2 -13499.999} C_VEL
LIN {X 0,Y 355.238,Z 413.731,A -85,B 0,C 180,E1 -13502.267,E2 -13502.267} C_VEL
LIN {X 0,Y 355.119,Z 413.748,A -85,B 0,C 180,E1 -13506.819,E2 -13506.819} C_VEL
LIN {X 0,Y 354.97,Z 413.765,A -85,B 0,C 180,E1 -13510.264,E2 -13510.264} C_VEL
LIN {X 0,Y 354.934,Z 413.77,A -85,B 0,C 180,E1 -13514.018,E2 -13514.018} C_VEL
LIN {X 0,Y 354.914,Z 413.772,A -85,B 0,C 180,E1 -13518.108,E2 -13518.108} C_VEL
LIN {X 0,Y 354.826,Z 413.783,A -85,B 0,C 180,E1 -13522.106,E2 -13522.106} C_VEL
LIN {X 0,Y 354.891,Z 413.775,A -85,B 0,C 180,E1 -13525.827,E2 -13525.827} C_VEL
LIN {X 0,Y 354.847,Z 413.781,A -85,B 0,C 180,E1 -13529.678,E2 -13529.678} C_VEL
LIN {X 0,Y 354.798,Z 413.787,A -85,B 0,C 180,E1 -13533.702,E2 -13533.702} C_VEL
LIN {X 0,Y 354.792,Z 413.789,A -85,B 0,C 180,E1 -13536.459,E2 -13536.459} C_VEL
LIN {X 0,Y 354.817,Z 413.785,A -85,B 0,C 180,E1 -13539.424,E2 -13539.424} C_VEL
LIN {X 0,Y 354.827,Z 413.788,A -85,B 0,C 180,E1 -13542.875,E2 -13542.875} C_VEL
LIN {X 0,Y 354.777,Z 413.79,A -85,B 0,C 180,E1 -13546.106,E2 -13546.106} C_VEL
LIN {X 0,Y 354.782,Z 413.79,A -85,B 0,C 180,E1 -13549.179,E2 -13549.179} C_VEL
LIN {X 0,Y 354.806,Z 413.79,A -85,B 0,C 180,E1 -13552.402,E2 -13552.402} C_VEL
LIN {X 0,Y 354.806,Z 413.788,A -85,B 0,C 180,E1 -13554.941,E2 -13554.941} C_VEL
LIN {X 0,Y 354.787,Z 413.793,A -85,B 0,C 180,E1 -13558.405,E2 -13558.405} C_VEL
LIN {X 0,Y 354.841,Z 413.781,A -85,B 0,C 180,E1 -13561.619,E2 -13561.619} C_VEL
LIN {X 0,Y 354.894,Z 413.778,A -85,B 0,C 180,E1 -13564.173,E2 -13564.173} C_VEL
LIN {X 0,Y 354.83,Z 413.784,A -85,B 0,C 180,E1 -13567.894,E2 -13567.894} C_VEL
LIN {X 0,Y 354.918,Z 413.777,A -85,B 0,C 180,E1 -13571.891,E2 -13571.891} C_VEL
LIN {X 0,Y 354.912,Z 413.816,A -85,B 0,C 180,E1 -13572.332,E2 -13572.332} C_VEL
LIN {X 0,Y 355.752,Z 416.384,A -85,B 0,C 180,E1 -13572.588,E2 -13572.588} C_VEL
LIN {X 0,Y 357.644,Z 418.563,A -85,B 0,C 180,E1 -13573.045,E2 -13573.045} C_VEL
LIN {X 0,Y 358.883,Z 419.509,A -85,B 0,C 180,E1 -13573.33,E2 -13573.33} C_VEL
LIN {X 0,Y 360.698,Z 422.456,A -85,B 0,C 180,E1 -13573.822,E2 -13573.822} C_VEL
LIN {X 0,Y 363.868,Z 425.405,A -85,B 0,C 180,E1 -13574.639,E2 -13574.639} C_VEL
LIN {X 0,Y 366.163,Z 428.515,A -85,B 0,C 180,E1 -13575.303,E2 -13575.303} C_VEL
LIN {X 0,Y 369.416,Z 431.287,A -85,B 0,C 180,E1 -13576.222,E2 -13576.222} C_VEL
LIN {X 0,Y 372.338,Z 434.832,A -85,B 0,C 180,E1 -13577.166,E2 -13577.166} C_VEL
LIN {X 0,Y 375.799,Z 437.611,A -85,B 0,C 180,E1 -13578.336,E2 -13578.336} C_VEL
LIN {X 0,Y 378.474,Z 440.74,A -85,B 0,C 180,E1 -13579.366,E2 -13579.366} C_VEL
LIN {X 0,Y 381.408,Z 443.015,A -85,B 0,C 180,E1 -13580.584,E2 -13580.584} C_VEL
LIN {X 0,Y 383.282,Z 444.111,A -85,B 0,C 180,E1 -13581.432,E2 -13581.432} C_VEL
LIN {X 0,Y 385.712,Z 447.137,A -85,B 0,C 180,E1 -13582.781,E2 -13582.781} C_VEL
LIN {X 0,Y 387.686,Z 448.933,A -85,B 0,C 180,E1 -13584.078,E2 -13584.078} C_VEL
LIN {X 0,Y 389.596,Z 450.122,A -85,B 0,C 180,E1 -13585.603,E2 -13585.603} C_VEL
LIN {X 0,Y 390.814,Z 450.439,A -85,B 0,C 180,E1 -13586.908,E2 -13586.908} C_VEL
LIN {X 0,Y 391.493,Z 450.613,A -85,B 0,C 180,E1 -13587.942,E2 -13587.942} C_VEL
LIN {X 0,Y 391.911,Z 450.646,A -85,B 0,C 180,E1 -13588.973,E2 -13588.973} C_VEL
LIN {X 0,Y 392.049,Z 450.672,A -85,B 0,C 180,E1 -13590,E2 -13590} C_VEL
LIN {X 0,Y 391.912,Z 450.65,A -85,B 0,C 180,E1 -13591.027,E2 -13591.027} C_VEL
LIN {X 0,Y 391.493,Z 450.606,A -85,B 0,C 180,E1 -13592.058,E2 -13592.058} C_VEL
LIN {X 0,Y 389.865,Z 450.224,A -85,B 0,C 180,E1 -13594.135,E2 -13594.135} C_VEL
LIN {X 0,Y 387.986,Z 449.124,A -85,B 0,C 180,E1 -13595.718,E2 -13595.718} C_VEL
LIN {X 0,Y 385.982,Z 447.456,A -85,B 0,C 180,E1 -13597.044,E2 -13597.044} C_VEL
LIN {X 0,Y 383.413,Z 444.308,A -85,B 0,C 180,E1 -13598.498,E2 -13598.498} C_VEL
LIN {X 0,Y 382.456,Z 443.553,A -85,B 0,C 180,E1 -13598.961,E2 -13598.961} C_VEL
LIN {X 0,Y 379.363,Z 441.556,A -85,B 0,C 180,E1 -13600.271,E2 -13600.271} C_VEL
LIN {X 0,Y 376.473,Z 438.528,A -85,B 0,C 180,E1 -13601.415,E2 -13601.415} C_VEL
LIN {X 0,Y 375.165,Z 436.97,A -85,B 0,C 180,E1 -13601.892,E2 -13601.892} C_VEL
LIN {X 0,Y 371.883,Z 434.407,A -85,B 0,C 180,E1 -13602.976,E2 -13602.976} C_VEL
LIN {X 0,Y 368.709,Z 430.568,A -85,B 0,C 180,E1 -13603.98,E2 -13603.98} C_VEL
LIN {X 0,Y 365.749,Z 428.067,A -85,B 0,C 180,E1 -13604.817,E2 -13604.817} C_VEL
LIN {X 0,Y 363.341,Z 424.761,A -85,B 0,C 180,E1 -13605.501,E2 -13605.501} C_VEL
LIN {X 0,Y 360.539,Z 422.269,A -85,B 0,C 180,E1 -13606.221,E2 -13606.221} C_VEL
LIN {X 0,Y 358.441,Z 419.088,A -85,B 0,C 180,E1 -13606.774,E2 -13606.774} C_VEL
LIN {X 0,Y 356.153,Z 417.025,A -85,B 0,C 180,E1 -13607.31,E2 -13607.31} C_VEL
LIN {X 0,Y 355.067,Z 414.681,A -85,B 0,C 180,E1 -13607.608,E2 -13607.608} C_VEL
LIN {X 0,Y 354.921,Z 413.777,A -85,B 0,C 180,E1 -13607.693,E2 -13607.693} C_VEL
LIN {X 0,Y 354.837,Z 413.786,A -85,B 0,C 180,E1 -13611.427,E2 -13611.427} C_VEL
LIN {X 0,Y 354.856,Z 413.779,A -85,B 0,C 180,E1 -13614.576,E2 -13614.576} C_VEL
LIN {X 0,Y 354.876,Z 413.779,A -85,B 0,C 180,E1 -13617.096,E2 -13617.096} C_VEL
LIN {X 0,Y 354.794,Z 413.789,A -85,B 0,C 180,E1 -13620.998,E2 -13620.998} C_VEL
LIN {X 0,Y 354.8,Z 413.79,A -85,B 0,C 180,E1 -13623.702,E2 -13623.702} C_VEL
LIN {X 0,Y 354.795,Z 413.787,A -85,B 0,C 180,E1 -13626.459,E2 -13626.459} C_VEL
LIN {X 0,Y 354.818,Z 413.79,A -85,B 0,C 180,E1 -13629.423,E2 -13629.423} C_VEL
LIN {X 0,Y 354.782,Z 413.79,A -85,B 0,C 180,E1 -13632.867,E2 -13632.867} C_VEL
LIN {X 0,Y 354.769,Z 413.79,A -85,B 0,C 180,E1 -13636.105,E2 -13636.105} C_VEL
LIN {X 0,Y 354.769,Z 413.792,A -85,B 0,C 180,E1 -13639.603,E2 -13639.603} C_VEL
LIN {X 0,Y 354.8,Z 413.786,A -85,B 0,C 180,E1 -13642.402,E2 -13642.402} C_VEL
LIN {X 0,Y 354.806,Z 413.786,A -85,B 0,C 180,E1 -13644.532,E2 -13644.532} C_VEL
LIN {X 0,Y 354.116,Z 413.877,A -85,B 0,C 180,E1 -13645.479,E2 -13645.479} C_VEL
LIN {X 0,Y 351.221,Z 414.238,A -85,B 0,C 180,E1 -13647.018,E2 -13647.018} C_VEL
LIN {X 0,Y 348.804,Z 414.533,A -85,B 0,C 180,E1 -13648.264,E2 -13648.264} C_VEL
LIN {X 0,Y 347.808,Z 414.661,A -85,B 0,C 180,E1 -13649.229,E2 -13649.229} C_VEL
LIN {X 0,Y 347.749,Z 414.665,A -85,B 0,C 180,E1 -13649.556,E2 -13649.556} C_VEL
LIN {X 0,Y 347.845,Z 414.656,A -85,B 0,C 180,E1 -13652.745,E2 -13652.745} C_VEL
LIN {X 0,Y 347.78,Z 414.661,A -85,B 0,C 180,E1 -13656.162,E2 -13656.162} C_VEL
LIN {X 0,Y 347.804,Z 414.657,A -85,B 0,C 180,E1 -13659.91,E2 -13659.91} C_VEL
LIN {X 0,Y 347.858,Z 414.653,A -85,B 0,C 180,E1 -13662.36,E2 -13662.36} C_VEL
LIN {X 0,Y 347.89,Z 414.647,A -85,B 0,C 180,E1 -13665.971,E2 -13665.971} C_VEL
LIN {X 0,Y 347.92,Z 414.643,A -85,B 0,C 180,E1 -13669.526,E2 -13669.526} C_VEL
LIN {X 0,Y 348.084,Z 414.625,A -85,B 0,C 180,E1 -13673.043,E2 -13673.043} C_VEL
LIN {X 0,Y 348.201,Z 414.607,A -85,B 0,C 180,E1 -13677.687,E2 -13677.687} C_VEL
LIN {X 0,Y 348.338,Z 414.591,A -85,B 0,C 180,E1 -13680.001,E2 -13680.001} C_VEL
LIN {X 0,Y 348.201,Z 414.612,A -85,B 0,C 180,E1 -13682.314,E2 -13682.314} C_VEL
LIN {X 0,Y 348.085,Z 414.624,A -85,B 0,C 180,E1 -13686.959,E2 -13686.959} C_VEL
LIN {X 0,Y 347.922,Z 414.648,A -85,B 0,C 180,E1 -13690.475,E2 -13690.475} C_VEL
LIN {X 0,Y 347.893,Z 414.651,A -85,B 0,C 180,E1 -13694.151,E2 -13694.151} C_VEL
LIN {X 0,Y 347.885,Z 414.653,A -85,B 0,C 180,E1 -13698.291,E2 -13698.291} C_VEL
LIN {X 0,Y 347.763,Z 414.664,A -85,B 0,C 180,E1 -13701.627,E2 -13701.627} C_VEL
LIN {X 0,Y 347.806,Z 414.658,A -85,B 0,C 180,E1 -13705.11,E2 -13705.11} C_VEL
LIN {X 0,Y 347.808,Z 414.66,A -85,B 0,C 180,E1 -13707.695,E2 -13707.695} C_VEL
LIN {X 0,Y 347.767,Z 414.666,A -85,B 0,C 180,E1 -13710.347,E2 -13710.347} C_VEL
LIN {X 0,Y 347.745,Z 414.671,A -85,B 0,C 180,E1 -13714.045,E2 -13714.045} C_VEL
LIN {X 0,Y 347.768,Z 414.668,A -85,B 0,C 180,E1 -13716.066,E2 -13716.066} C_VEL
LIN {X 0,Y 348.181,Z 417.494,A -85,B 0,C 180,E1 -13719.914,E2 -13719.914} C_VEL
LIN {X 0,Y 348.622,Z 420.426,A -85,B 0,C 180,E1 -13723.471,E2 -13723.471} C_VEL
LIN {X 0,Y 348.826,Z 423.387,A -85,B 0,C 180,E1 -13726.764,E2 -13726.764} C_VEL
LIN {X 0,Y 348.669,Z 426.406,A -85,B 0,C 180,E1 -13729.834,E2 -13729.834} C_VEL
LIN {X 0,Y 348.34,Z 429.468,A -85,B 0,C 180,E1 -13732.753,E2 -13732.753} C_VEL
LIN {X 0,Y 347.946,Z 432.958,A -85,B 0,C 180,E1 -13735.909,E2 -13735.909} C_VEL
LIN {X 0,Y 347.449,Z 437.274,A -85,B 0,C 180,E1 -13739.624,E2 -13739.624} C_VEL
LIN {X 0,Y 347.011,Z 442.041,A -85,B 0,C 180,E1 -13743.541,E2 -13743.541} C_VEL
LIN {X 0,Y 346.758,Z 445.23,A -85,B 0,C 180,E1 -13746.087,E2 -13746.087} C_VEL
LIN {X 0,Y 346.543,Z 449.027,A -85,B 0,C 180,E1 -13749.084,E2 -13749.084} C_VEL
LIN {X 0,Y 349.599,Z 463.004,A -85,B 0,C 180,E1 -13749.828,E2 -13749.828} C_VEL
LIN {X 0,Y 351.706,Z 475.814,A -85,B 0,C 180,E1 -13750.727,E2 -13750.727} C_VEL
LIN {X 0,Y 352.799,Z 485.677,A -85,B 0,C 180,E1 -13751.565,E2 -13751.565} C_VEL
LIN {X 0,Y 352.285,Z 493.61,A -85,B 0,C 180,E1 -13752.288,E2 -13752.288} C_VEL
LIN {X 0,Y 351.12,Z 503.905,A -85,B 0,C 180,E1 -13753.428,E2 -13753.428} C_VEL
LIN {X 0,Y 350.262,Z 511.212,A -85,B 0,C 180,E1 -13754.392,E2 -13754.392} C_VEL
LIN {X 0,Y 349.304,Z 519.656,A -85,B 0,C 180,E1 -13755.732,E2 -13755.732} C_VEL
LIN {X 0,Y 348.567,Z 525.859,A -85,B 0,C 180,E1 -13756.89,E2 -13756.89} C_VEL
LIN {X 0,Y 347.725,Z 532.395,A -85,B 0,C 180,E1 -13758.34,E2 -13758.34} C_VEL
LIN {X 0,Y 347.272,Z 536.899,A -85,B 0,C 180,E1 -13759.506,E2 -13759.506} C_VEL
LIN {X 0,Y 346.728,Z 542.392,A -85,B 0,C 180,E1 -13761.256,E2 -13761.256} C_VEL
LIN {X 0,Y 346.346,Z 546.716,A -85,B 0,C 180,E1 -13763.007,E2 -13763.007} C_VEL
LIN {X 0,Y 346.203,Z 549.084,A -85,B 0,C 180,E1 -13764.175,E2 -13764.175} C_VEL
LIN {X 0,Y 346.177,Z 550.885,A -85,B 0,C 180,E1 -13765.342,E2 -13765.342} C_VEL
LIN {X 0,Y 346.085,Z 553.33,A -85,B 0,C 180,E1 -13767.672,E2 -13767.672} C_VEL
LIN {X 0,Y 346.104,Z 553.92,A -85,B 0,C 180,E1 -13768.836,E2 -13768.836} C_VEL
LIN {X 0,Y 346.164,Z 554.076,A -85,B 0,C 180,E1 -13770,E2 -13770} C_VEL
LIN {X 0,Y 346.104,Z 553.92,A -85,B 0,C 180,E1 -13771.164,E2 -13771.164} C_VEL
LIN {X 0,Y 346.085,Z 553.33,A -85,B 0,C 180,E1 -13772.328,E2 -13772.328} C_VEL
LIN {X 0,Y 346.177,Z 550.885,A -85,B 0,C 180,E1 -13774.658,E2 -13774.658} C_VEL
LIN {X 0,Y 346.248,Z 547.934,A -85,B 0,C 180,E1 -13776.409,E2 -13776.409} C_VEL
LIN {X 0,Y 346.575,Z 543.945,A -85,B 0,C 180,E1 -13778.16,E2 -13778.16} C_VEL
LIN {X 0,Y 347.048,Z 538.814,A -85,B 0,C 180,E1 -13779.912,E2 -13779.912} C_VEL
LIN {X 0,Y 347.591,Z 533.551,A -85,B 0,C 180,E1 -13781.369,E2 -13781.369} C_VEL
LIN {X 0,Y 348.383,Z 527.235,A -85,B 0,C 180,E1 -13782.821,E2 -13782.821} C_VEL
LIN {X 0,Y 349.126,Z 521.284,A -85,B 0,C 180,E1 -13783.978,E2 -13783.978} C_VEL
LIN {X 0,Y 350.075,Z 513.108,A -85,B 0,C 180,E1 -13785.322,E2 -13785.322} C_VEL
LIN {X 0,Y 350.934,Z 505.038,A -85,B 0,C 180,E1 -13786.431,E2 -13786.431} C_VEL
LIN {X 0,Y 351.947,Z 496.312,A -85,B 0,C 180,E1 -13787.429,E2 -13787.429} C_VEL
LIN {X 0,Y 352.843,Z 487.315,A -85,B 0,C 180,E1 -13788.283,E2 -13788.283} C_VEL
LIN {X 0,Y 352.085,Z 478.921,A -85,B 0,C 180,E1 -13789.019,E2 -13789.019} C_VEL
LIN {X 0,Y 350.828,Z 470.182,A -85,B 0,C 180,E1 -13789.688,E2 -13789.688} C_VEL
LIN {X 0,Y 348.949,Z 459.953,A -85,B 0,C 180,E1 -13790.344,E2 -13790.344} C_VEL
LIN {X 0,Y 346.56,Z 449.006,A -85,B 0,C 180,E1 -13790.932,E2 -13790.932} C_VEL
LIN {X 0,Y 346.855,Z 443.614,A -85,B 0,C 180,E1 -13795.182,E2 -13795.182} C_VEL
LIN {X 0,Y 347.298,Z 438.845,A -85,B 0,C 180,E1 -13799.056,E2 -13799.056} C_VEL
LIN {X 0,Y 347.671,Z 435.474,A -85,B 0,C 180,E1 -13801.895,E2 -13801.895} C_VEL
LIN {X 0,Y 348.182,Z 431.012,A -85,B 0,C 180,E1 -13805.828,E2 -13805.828} C_VEL
LIN {X 0,Y 348.53,Z 427.929,A -85,B 0,C 180,E1 -13808.689,E2 -13808.689} C_VEL
LIN {X 0,Y 348.807,Z 424.765,A -85,B 0,C 180,E1 -13811.797,E2 -13811.797} C_VEL
LIN {X 0,Y 348.77,Z 421.868,A -85,B 0,C 180,E1 -13814.851,E2 -13814.851} C_VEL
LIN {X 0,Y 348.384,Z 418.925,A -85,B 0,C 180,E1 -13818.279,E2 -13818.279} C_VEL
LIN {X 0,Y 347.945,Z 416.062,A -85,B 0,C 180,E1 -13821.974,E2 -13821.974} C_VEL
LIN {X 0,Y 347.786,Z 414.667,A -85,B 0,C 180,E1 -13824.124,E2 -13824.124} C_VEL
LIN {X 0,Y 347.76,Z 414.667,A -85,B 0,C 180,E1 -13828.301,E2 -13828.301} C_VEL
LIN {X 0,Y 347.802,Z 414.658,A -85,B 0,C 180,E1 -13830.989,E2 -13830.989} C_VEL
LIN {X 0,Y 347.827,Z 414.658,A -85,B 0,C 180,E1 -13833.607,E2 -13833.607} C_VEL
LIN {X 0,Y 347.78,Z 414.664,A -85,B 0,C 180,E1 -13836.161,E2 -13836.161} C_VEL
LIN {X 0,Y 347.801,Z 414.663,A -85,B 0,C 180,E1 -13839.908,E2 -13839.908} C_VEL
LIN {X 0,Y 347.861,Z 414.652,A -85,B 0,C 180,E1 -13842.358,E2 -13842.358} C_VEL
LIN {X 0,Y 347.892,Z 414.65,A -85,B 0,C 180,E1 -13845.97,E2 -13845.97} C_VEL
LIN {X 0,Y 347.922,Z 414.648,A -85,B 0,C 180,E1 -13849.525,E2 -13849.525} C_VEL
LIN {X 0,Y 348.085,Z 414.624,A -85,B 0,C 180,E1 -13853.041,E2 -13853.041} C_VEL
LIN {X 0,Y 348.201,Z 414.612,A -85,B 0,C 180,E1 -13857.686,E2 -13857.686} C_VEL
LIN {X 0,Y 348.338,Z 414.591,A -85,B 0,C 180,E1 -13859.999,E2 -13859.999} C_VEL
LIN {X 0,Y 348.201,Z 414.607,A -85,B 0,C 180,E1 -13862.313,E2 -13862.313} C_VEL
LIN {X 0,Y 348.084,Z 414.625,A -85,B 0,C 180,E1 -13866.957,E2 -13866.957} C_VEL
LIN {X 0,Y 347.92,Z 414.643,A -85,B 0,C 180,E1 -13870.474,E2 -13870.474} C_VEL
LIN {X 0,Y 347.891,Z 414.647,A -85,B 0,C 180,E1 -13874.149,E2 -13874.149} C_VEL
LIN {X 0,Y 347.883,Z 414.648,A -85,B 0,C 180,E1 -13878.29,E2 -13878.29} C_VEL
LIN {X 0,Y 347.78,Z 414.662,A -85,B 0,C 180,E1 -13881.635,E2 -13881.635} C_VEL
LIN {X 0,Y 347.805,Z 414.663,A -85,B 0,C 180,E1 -13885.108,E2 -13885.108} C_VEL
LIN {X 0,Y 347.804,Z 414.658,A -85,B 0,C 180,E1 -13887.694,E2 -13887.694} C_VEL
LIN {X 0,Y 347.757,Z 414.664,A -85,B 0,C 180,E1 -13890.346,E2 -13890.346} C_VEL
LIN {X 0,Y 347.737,Z 414.668,A -85,B 0,C 180,E1 -13894.464,E2 -13894.464} C_VEL
LIN {X 0,Y 347.769,Z 414.662,A -85,B 0,C 180,E1 -13897.989,E2 -13897.989} C_VEL
LIN {X 0,Y 347.777,Z 414.661,A -85,B 0,C 180,E1 -13901.609,E2 -13901.609} C_VEL
LIN {X 0,Y 347.789,Z 414.663,A -85,B 0,C 180,E1 -13905.012,E2 -13905.012} C_VEL
LIN {X 0,Y 347.744,Z 414.668,A -85,B 0,C 180,E1 -13908.397,E2 -13908.397} C_VEL
LIN {X 0,Y 347.771,Z 414.663,A -85,B 0,C 180,E1 -13912.011,E2 -13912.011} C_VEL
LIN {X 0,Y 347.738,Z 414.666,A -85,B 0,C 180,E1 -13915.536,E2 -13915.536} C_VEL
LIN {X 0,Y 347.739,Z 414.67,A -85,B 0,C 180,E1 -13918.301,E2 -13918.301} C_VEL
LIN {X 0,Y 347.773,Z 414.663,A -85,B 0,C 180,E1 -13920.988,E2 -13920.988} C_VEL
LIN {X 0,Y 347.826,Z 414.655,A -85,B 0,C 180,E1 -13923.608,E2 -13923.608} C_VEL
LIN {X 0,Y 347.784,Z 414.664,A -85,B 0,C 180,E1 -13926.162,E2 -13926.162} C_VEL
LIN {X 0,Y 347.813,Z 414.661,A -85,B 0,C 180,E1 -13929.91,E2 -13929.91} C_VEL
LIN {X 0,Y 347.839,Z 414.659,A -85,B 0,C 180,E1 -13931.025,E2 -13931.025} C_VEL
LIN {X 0,Y 348.762,Z 417.38,A -85,B 0,C 180,E1 -13931.28,E2 -13931.28} C_VEL
LIN {X 0,Y 350.818,Z 419.58,A -85,B 0,C 180,E1 -13931.728,E2 -13931.728} C_VEL
LIN {X 0,Y 351.518,Z 420.236,A -85,B 0,C 180,E1 -13931.881,E2 -13931.881} C_VEL
LIN {X 0,Y 353.708,Z 423.581,A -85,B 0,C 180,E1 -13932.398,E2 -13932.398} C_VEL
LIN {X 0,Y 356.055,Z 425.832,A -85,B 0,C 180,E1 -13932.95,E2 -13932.95} C_VEL
LIN {X 0,Y 358.554,Z 429.125,A -85,B 0,C 180,E1 -13933.57,E2 -13933.57} C_VEL
LIN {X 0,Y 361.248,Z 431.686,A -85,B 0,C 180,E1 -13934.26,E2 -13934.26} C_VEL
LIN {X 0,Y 364.316,Z 435.303,A -85,B 0,C 180,E1 -13935.083,E2 -13935.083} C_VEL
LIN {X 0,Y 367.162,Z 437.793,A -85,B 0,C 180,E1 -13935.896,E2 -13935.896} C_VEL
LIN {X 0,Y 370.391,Z 441.421,A -85,B 0,C 180,E1 -13936.883,E2 -13936.883} C_VEL
LIN {X 0,Y 374.051,Z 444.36,A -85,B 0,C 180,E1 -13938.073,E2 -13938.073} C_VEL
LIN {X 0,Y 376.844,Z 447.451,A -85,B 0,C 180,E1 -13939.116,E2 -13939.116} C_VEL
LIN {X 0,Y 380.1,Z 449.908,A -85,B 0,C 180,E1 -13940.421,E2 -13940.421} C_VEL
LIN {X 0,Y 382.04,Z 451.164,A -85,B 0,C 180,E1 -13941.288,E2 -13941.288} C_VEL
LIN {X 0,Y 384.763,Z 454.33,A -85,B 0,C 180,E1 -13942.763,E2 -13942.763} C_VEL
LIN {X 0,Y 387.068,Z 456.228,A -85,B 0,C 180,E1 -13944.269,E2 -13944.269} C_VEL
LIN {X 0,Y 388.978,Z 457.245,A -85,B 0,C 180,E1 -13945.856,E2 -13945.856} C_VEL
LIN {X 0,Y 389.939,Z 457.473,A -85,B 0,C 180,E1 -13946.901,E2 -13946.901} C_VEL
LIN {X 0,Y 390.625,Z 457.63,A -85,B 0,C 180,E1 -13947.938,E2 -13947.938} C_VEL
LIN {X 0,Y 391.046,Z 457.675,A -85,B 0,C 180,E1 -13948.97,E2 -13948.97} C_VEL
LIN {X 0,Y 391.184,Z 457.719,A -85,B 0,C 180,E1 -13950,E2 -13950} C_VEL
LIN {X 0,Y 391.046,Z 457.679,A -85,B 0,C 180,E1 -13951.03,E2 -13951.03} C_VEL
LIN {X 0,Y 390.621,Z 457.652,A -85,B 0,C 180,E1 -13952.062,E2 -13952.062} C_VEL
LIN {X 0,Y 389.525,Z 457.374,A -85,B 0,C 180,E1 -13953.61,E2 -13953.61} C_VEL
LIN {X 0,Y 387.765,Z 456.677,A -85,B 0,C 180,E1 -13955.199,E2 -13955.199} C_VEL
LIN {X 0,Y 385.509,Z 455.055,A -85,B 0,C 180,E1 -13956.768,E2 -13956.768} C_VEL
LIN {X 0,Y 382.719,Z 452.057,A -85,B 0,C 180,E1 -13958.361,E2 -13958.361} C_VEL
LIN {X 0,Y 381.489,Z 450.607,A -85,B 0,C 180,E1 -13958.984,E2 -13958.984} C_VEL
LIN {X 0,Y 378.16,Z 448.582,A -85,B 0,C 180,E1 -13960.372,E2 -13960.372} C_VEL
LIN {X 0,Y 374.823,Z 445.375,A -85,B 0,C 180,E1 -13961.64,E2 -13961.64} C_VEL
LIN {X 0,Y 373.241,Z 443.582,A -85,B 0,C 180,E1 -13962.213,E2 -13962.213} C_VEL
LIN {X 0,Y 369.641,Z 440.69,A -85,B 0,C 180,E1 -13963.353,E2 -13963.353} C_VEL
LIN {X 0,Y 366.323,Z 436.916,A -85,B 0,C 180,E1 -13964.348,E2 -13964.348} C_VEL
LIN {X 0,Y 363.18,Z 434.15,A -85,B 0,C 180,E1 -13965.219,E2 -13965.219} C_VEL
LIN {X 0,Y 360.502,Z 430.862,A -85,B 0,C 180,E1 -13965.94,E2 -13965.94} C_VEL
LIN {X 0,Y 357.446,Z 427.911,A -85,B 0,C 180,E1 -13966.695,E2 -13966.695} C_VEL
LIN {X 0,Y 355.394,Z 425.109,A -85,B 0,C 180,E1 -13967.209,E2 -13967.209} C_VEL
LIN {X 0,Y 352.737,Z 422.378,A -85,B 0,C 180,E1 -13967.823,E2 -13967.823} C_VEL
LIN {X 0,Y 351.102,Z 419.768,A -85,B 0,C 180,E1 -13968.213,E2 -13968.213} C_VEL
LIN {X 0,Y 348.923,Z 417.616,A -85,B 0,C 180,E1 -13968.683,E2 -13968.683} C_VEL
LIN {X 0,Y 347.945,Z 415.35,A -85,B 0,C 180,E1 -13968.931,E2 -13968.931} C_VEL
LIN {X 0,Y 347.828,Z 414.66,A -85,B 0,C 180,E1 -13969.014,E2 -13969.014} C_VEL
LIN {X 0,Y 347.771,Z 414.662,A -85,B 0,C 180,E1 -13972.579,E2 -13972.579} C_VEL
LIN {X 0,Y 347.807,Z 414.659,A -85,B 0,C 180,E1 -13975.108,E2 -13975.108} C_VEL
LIN {X 0,Y 347.803,Z 414.663,A -85,B 0,C 180,E1 -13977.694,E2 -13977.694} C_VEL
LIN {X 0,Y 347.743,Z 414.666,A -85,B 0,C 180,E1 -13980.348,E2 -13980.348} C_VEL
LIN {X 0,Y 347.742,Z 414.667,A -85,B 0,C 180,E1 -13984.044,E2 -13984.044} C_VEL
LIN {X 0,Y 347.759,Z 414.669,A -85,B 0,C 180,E1 -13987.32,E2 -13987.32} C_VEL
LIN {X 0,Y 347.726,Z 414.667,A -85,B 0,C 180,E1 -13990.297,E2 -13990.297} C_VEL
LIN {X 0,Y 347.719,Z 414.673,A -85,B 0,C 180,E1 -13993.407,E2 -13993.407} C_VEL
LIN {X 0,Y 347.72,Z 414.669,A -85,B 0,C 180,E1 -13996.686,E2 -13996.686} C_VEL
LIN {X 0,Y 347.74,Z 414.666,A -85,B 0,C 180,E1 -14000.173,E2 -14000.173} C_VEL
LIN {X 0,Y 347.755,Z 414.666,A -85,B 0,C 180,E1 -14002.679,E2 -14002.679} C_VEL
LIN {X 0,Y 347.741,Z 414.666,A -85,B 0,C 180,E1 -14005.956,E2 -14005.956} C_VEL
LIN {X 0,Y 347.749,Z 414.665,A -85,B 0,C 180,E1 -14009.556,E2 -14009.556} C_VEL
LIN {X 0,Y 347.142,Z 414.745,A -85,B 0,C 180,E1 -14010.524,E2 -14010.524} C_VEL
LIN {X 0,Y 344.318,Z 415.097,A -85,B 0,C 180,E1 -14012.098,E2 -14012.098} C_VEL
LIN {X 0,Y 341.888,Z 415.397,A -85,B 0,C 180,E1 -14013.373,E2 -14013.373} C_VEL
LIN {X 0,Y 340.84,Z 415.526,A -85,B 0,C 180,E1 -14014.359,E2 -14014.359} C_VEL
LIN {X 0,Y 340.753,Z 415.537,A -85,B 0,C 180,E1 -14014.693,E2 -14014.693} C_VEL
LIN {X 0,Y 340.734,Z 415.539,A -85,B 0,C 180,E1 -14018.207,E2 -14018.207} C_VEL
LIN {X 0,Y 340.85,Z 415.524,A -85,B 0,C 180,E1 -14021.985,E2 -14021.985} C_VEL
LIN {X 0,Y 340.862,Z 415.522,A -85,B 0,C 180,E1 -14025.705,E2 -14025.705} C_VEL
LIN {X 0,Y 340.863,Z 415.523,A -85,B 0,C 180,E1 -14029.307,E2 -14029.307} C_VEL
LIN {X 0,Y 341.052,Z 415.502,A -85,B 0,C 180,E1 -14032.898,E2 -14032.898} C_VEL
LIN {X 0,Y 341.163,Z 415.482,A -85,B 0,C 180,E1 -14037.639,E2 -14037.639} C_VEL
LIN {X 0,Y 341.289,Z 415.469,A -85,B 0,C 180,E1 -14040.001,E2 -14040.001} C_VEL
LIN {X 0,Y 341.163,Z 415.489,A -85,B 0,C 180,E1 -14042.362,E2 -14042.362} C_VEL
LIN {X 0,Y 341.053,Z 415.499,A -85,B 0,C 180,E1 -14047.103,E2 -14047.103} C_VEL
LIN {X 0,Y 340.864,Z 415.525,A -85,B 0,C 180,E1 -14050.695,E2 -14050.695} C_VEL
LIN {X 0,Y 340.857,Z 415.529,A -85,B 0,C 180,E1 -14054.326,E2 -14054.326} C_VEL
LIN {X 0,Y 340.832,Z 415.53,A -85,B 0,C 180,E1 -14058.467,E2 -14058.467} C_VEL
LIN {X 0,Y 340.713,Z 415.544,A -85,B 0,C 180,E1 -14061.843,E2 -14061.843} C_VEL
LIN {X 0,Y 340.768,Z 415.537,A -85,B 0,C 180,E1 -14065.665,E2 -14065.665} C_VEL
LIN {X 0,Y 340.738,Z 415.542,A -85,B 0,C 180,E1 -14068.321,E2 -14068.321} C_VEL
LIN {X 0,Y 340.712,Z 415.542,A -85,B 0,C 180,E1 -14071.044,E2 -14071.044} C_VEL
LIN {X 0,Y 340.715,Z 415.545,A -85,B 0,C 180,E1 -14075.28,E2 -14075.28} C_VEL
LIN {X 0,Y 340.808,Z 416.226,A -85,B 0,C 180,E1 -14076.729,E2 -14076.729} C_VEL
LIN {X 0,Y 341.214,Z 418.921,A -85,B 0,C 180,E1 -14080.353,E2 -14080.353} C_VEL
LIN {X 0,Y 341.619,Z 421.885,A -85,B 0,C 180,E1 -14083.943,E2 -14083.943} C_VEL
LIN {X 0,Y 341.76,Z 423.69,A -85,B 0,C 180,E1 -14086.034,E2 -14086.034} C_VEL
LIN {X 0,Y 341.706,Z 426.339,A -85,B 0,C 180,E1 -14088.842,E2 -14088.842} C_VEL
LIN {X 0,Y 341.413,Z 429.392,A -85,B 0,C 180,E1 -14091.864,E2 -14091.864} C_VEL
LIN {X 0,Y 340.931,Z 433.331,A -85,B 0,C 180,E1 -14095.545,E2 -14095.545} C_VEL
LIN {X 0,Y 340.473,Z 437.151,A -85,B 0,C 180,E1 -14098.933,E2 -14098.933} C_VEL
LIN {X 0,Y 339.976,Z 441.892,A -85,B 0,C 180,E1 -14102.95,E2 -14102.95} C_VEL
LIN {X 0,Y 339.742,Z 445.085,A -85,B 0,C 180,E1 -14105.562,E2 -14105.562} C_VEL
LIN {X 0,Y 339.487,Z 448.855,A -85,B 0,C 180,E1 -14108.627,E2 -14108.627} C_VEL
LIN {X 0,Y 342.704,Z 463.407,A -85,B 0,C 180,E1 -14109.434,E2 -14109.434} C_VEL
LIN {X 0,Y 344.713,Z 475.442,A -85,B 0,C 180,E1 -14110.308,E2 -14110.308} C_VEL
LIN {X 0,Y 345.914,Z 485.475,A -85,B 0,C 180,E1 -14111.184,E2 -14111.184} C_VEL
LIN {X 0,Y 345.7,Z 491.994,A -85,B 0,C 180,E1 -14111.786,E2 -14111.786} C_VEL
LIN {X 0,Y 344.432,Z 502.573,A -85,B 0,C 180,E1 -14112.944,E2 -14112.944} C_VEL
LIN {X 0,Y 343.287,Z 511.861,A -85,B 0,C 180,E1 -14114.201,E2 -14114.201} C_VEL
LIN {X 0,Y 342.382,Z 519.458,A -85,B 0,C 180,E1 -14115.437,E2 -14115.437} C_VEL
LIN {X 0,Y 341.631,Z 525.661,A -85,B 0,C 180,E1 -14116.619,E2 -14116.619} C_VEL
LIN {X 0,Y 340.744,Z 532.197,A -85,B 0,C 180,E1 -14118.097,E2 -14118.097} C_VEL
LIN {X 0,Y 340.259,Z 536.701,A -85,B 0,C 180,E1 -14119.287,E2 -14119.287} C_VEL
LIN {X 0,Y 339.692,Z 542.194,A -85,B 0,C 180,E1 -14121.074,E2 -14121.074} C_VEL
LIN {X 0,Y 339.277,Z 546.519,A -85,B 0,C 180,E1 -14122.861,E2 -14122.861} C_VEL
LIN {X 0,Y 339.114,Z 549.033,A -85,B 0,C 180,E1 -14124.148,E2 -14124.148} C_VEL
LIN {X 0,Y 339.073,Z 552.076,A -85,B 0,C 180,E1 -14126.435,E2 -14126.435} C_VEL
LIN {X 0,Y 339,Z 553.133,A -85,B 0,C 180,E1 -14127.624,E2 -14127.624} C_VEL
LIN {X 0,Y 339.007,Z 553.723,A -85,B 0,C 180,E1 -14128.812,E2 -14128.812} C_VEL
LIN {X 0,Y 339.066,Z 553.879,A -85,B 0,C 180,E1 -14130,E2 -14130} C_VEL
LIN {X 0,Y 339.007,Z 553.723,A -85,B 0,C 180,E1 -14131.188,E2 -14131.188} C_VEL
LIN {X 0,Y 339,Z 553.133,A -85,B 0,C 180,E1 -14132.376,E2 -14132.376} C_VEL
LIN {X 0,Y 339.078,Z 550.687,A -85,B 0,C 180,E1 -14134.756,E2 -14134.756} C_VEL
LIN {X 0,Y 339.17,Z 547.735,A -85,B 0,C 180,E1 -14136.544,E2 -14136.544} C_VEL
LIN {X 0,Y 339.535,Z 543.748,A -85,B 0,C 180,E1 -14138.331,E2 -14138.331} C_VEL
LIN {X 0,Y 340.041,Z 538.617,A -85,B 0,C 180,E1 -14140.118,E2 -14140.118} C_VEL
LIN {X 0,Y 340.598,Z 533.353,A -85,B 0,C 180,E1 -14141.606,E2 -14141.606} C_VEL
LIN {X 0,Y 341.435,Z 527.037,A -85,B 0,C 180,E1 -14143.086,E2 -14143.086} C_VEL
LIN {X 0,Y 342.197,Z 521.085,A -85,B 0,C 180,E1 -14144.267,E2 -14144.267} C_VEL
LIN {X 0,Y 343.172,Z 513.09,A -85,B 0,C 180,E1 -14145.609,E2 -14145.609} C_VEL
LIN {X 0,Y 344.103,Z 504.841,A -85,B 0,C 180,E1 -14146.767,E2 -14146.767} C_VEL
LIN {X 0,Y 345.148,Z 496.114,A -85,B 0,C 180,E1 -14147.784,E2 -14147.784} C_VEL
LIN {X 0,Y 345.965,Z 488.75,A -85,B 0,C 180,E1 -14148.506,E2 -14148.506} C_VEL
LIN {X 0,Y 345.348,Z 480.615,A -85,B 0,C 180,E1 -14149.26,E2 -14149.26} C_VEL
LIN {X 0,Y 344.069,Z 471.27,A -85,B 0,C 180,E1 -14150.014,E2 -14150.014} C_VEL
LIN {X 0,Y 342.017,Z 460.101,A -85,B 0,C 180,E1 -14150.76,E2 -14150.76} C_VEL
LIN {X 0,Y 339.487,Z 448.855,A -85,B 0,C 180,E1 -14151.373,E2 -14151.373} C_VEL
LIN {X 0,Y 339.737,Z 445.008,A -85,B 0,C 180,E1 -14154.464,E2 -14154.464} C_VEL
LIN {X 0,Y 340.112,Z 440.29,A -85,B 0,C 180,E1 -14158.376,E2 -14158.376} C_VEL
LIN {X 0,Y 340.641,Z 435.816,A -85,B 0,C 180,E1 -14162.23,E2 -14162.23} C_VEL
LIN {X 0,Y 341.009,Z 432.467,A -85,B 0,C 180,E1 -14165.243,E2 -14165.243} C_VEL
LIN {X 0,Y 341.46,Z 428.962,A -85,B 0,C 180,E1 -14168.544,E2 -14168.544} C_VEL
LIN {X 0,Y 341.707,Z 426.333,A -85,B 0,C 180,E1 -14171.158,E2 -14171.158} C_VEL
LIN {X 0,Y 341.746,Z 423.328,A -85,B 0,C 180,E1 -14174.362,E2 -14174.362} C_VEL
LIN {X 0,Y 341.395,Z 420.325,A -85,B 0,C 180,E1 -14177.824,E2 -14177.824} C_VEL
LIN {X 0,Y 341.133,Z 418.401,A -85,B 0,C 180,E1 -14180.307,E2 -14180.307} C_VEL
LIN {X 0,Y 340.791,Z 416.036,A -85,B 0,C 180,E1 -14183.539,E2 -14183.539} C_VEL
LIN {X 0,Y 340.715,Z 415.549,A -85,B 0,C 180,E1 -14184.72,E2 -14184.72} C_VEL
LIN {X 0,Y 340.712,Z 415.543,A -85,B 0,C 180,E1 -14188.956,E2 -14188.956} C_VEL
LIN {X 0,Y 340.776,Z 415.535,A -85,B 0,C 180,E1 -14192.473,E2 -14192.473} C_VEL
LIN {X 0,Y 340.75,Z 415.541,A -85,B 0,C 180,E1 -14195.637,E2 -14195.637} C_VEL
LIN {X 0,Y 340.729,Z 415.542,A -85,B 0,C 180,E1 -14199.472,E2 -14199.472} C_VEL
LIN {X 0,Y 340.852,Z 415.528,A -85,B 0,C 180,E1 -14201.983,E2 -14201.983} C_VEL
LIN {X 0,Y 340.864,Z 415.528,A -85,B 0,C 180,E1 -14205.704,E2 -14205.704} C_VEL
LIN {X 0,Y 340.864,Z 415.525,A -85,B 0,C 180,E1 -14209.305,E2 -14209.305} C_VEL
LIN {X 0,Y 341.053,Z 415.499,A -85,B 0,C 180,E1 -14212.897,E2 -14212.897} C_VEL
LIN {X 0,Y 341.163,Z 415.489,A -85,B 0,C 180,E1 -14217.638,E2 -14217.638} C_VEL
LIN {X 0,Y 341.289,Z 415.469,A -85,B 0,C 180,E1 -14219.999,E2 -14219.999} C_VEL
LIN {X 0,Y 341.163,Z 415.482,A -85,B 0,C 180,E1 -14222.361,E2 -14222.361} C_VEL
LIN {X 0,Y 341.052,Z 415.502,A -85,B 0,C 180,E1 -14227.102,E2 -14227.102} C_VEL
LIN {X 0,Y 340.863,Z 415.523,A -85,B 0,C 180,E1 -14230.693,E2 -14230.693} C_VEL
LIN {X 0,Y 340.855,Z 415.523,A -85,B 0,C 180,E1 -14234.324,E2 -14234.324} C_VEL
LIN {X 0,Y 340.829,Z 415.527,A -85,B 0,C 180,E1 -14238.466,E2 -14238.466} C_VEL
LIN {X 0,Y 340.746,Z 415.537,A -85,B 0,C 180,E1 -14241.857,E2 -14241.857} C_VEL
LIN {X 0,Y 340.765,Z 415.535,A -85,B 0,C 180,E1 -14245.664,E2 -14245.664} C_VEL
LIN {X 0,Y 340.735,Z 415.539,A -85,B 0,C 180,E1 -14248.319,E2 -14248.319} C_VEL
LIN {X 0,Y 340.696,Z 415.548,A -85,B 0,C 180,E1 -14251.044,E2 -14251.044} C_VEL
LIN {X 0,Y 340.711,Z 415.544,A -85,B 0,C 180,E1 -14255.279,E2 -14255.279} C_VEL
LIN {X 0,Y 340.711,Z 415.543,A -85,B 0,C 180,E1 -14258.388,E2 -14258.388} C_VEL
LIN {X 0,Y 340.718,Z 415.542,A -85,B 0,C 180,E1 -14261.304,E2 -14261.304} C_VEL
LIN {X 0,Y 340.714,Z 415.545,A -85,B 0,C 180,E1 -14264.533,E2 -14264.533} C_VEL
LIN {X 0,Y 340.68,Z 415.551,A -85,B 0,C 180,E1 -14268.691,E2 -14268.691} C_VEL
LIN {X 0,Y 340.729,Z 415.539,A -85,B 0,C 180,E1 -14271.773,E2 -14271.773} C_VEL
LIN {X 0,Y 340.717,Z 415.541,A -85,B 0,C 180,E1 -14275.596,E2 -14275.596} C_VEL
LIN {X 0,Y 340.692,Z 415.546,A -85,B 0,C 180,E1 -14278.956,E2 -14278.956} C_VEL
LIN {X 0,Y 340.798,Z 415.532,A -85,B 0,C 180,E1 -14283.02,E2 -14283.02} C_VEL
LIN {X 0,Y 340.751,Z 415.537,A -85,B 0,C 180,E1 -14285.639,E2 -14285.639} C_VEL
LIN {X 0,Y 340.775,Z 415.537,A -85,B 0,C 180,E1 -14289.76,E2 -14289.76} C_VEL
LIN {X 0,Y 340.766,Z 415.538,A -85,B 0,C 180,E1 -14289.83,E2 -14289.83} C_VEL
LIN {X 0,Y 341.795,Z 418.434,A -85,B 0,C 180,E1 -14290.105,E2 -14290.105} C_VEL
LIN {X 0,Y 344.235,Z 421.101,A -85,B 0,C 180,E1 -14290.593,E2 -14290.593} C_VEL
LIN {X 0,Y 346.385,Z 424.317,A -85,B 0,C 180,E1 -14291.057,E2 -14291.057} C_VEL
LIN {X 0,Y 348.434,Z 426.493,A -85,B 0,C 180,E1 -14291.494,E2 -14291.494} C_VEL
LIN {X 0,Y 351.293,Z 430.162,A -85,B 0,C 180,E1 -14292.145,E2 -14292.145} C_VEL
LIN {X 0,Y 353.191,Z 432.043,A -85,B 0,C 180,E1 -14292.561,E2 -14292.561} C_VEL
LIN {X 0,Y 356.394,Z 435.839,A -85,B 0,C 180,E1 -14293.344,E2 -14293.344} C_VEL
LIN {X 0,Y 358.684,Z 437.944,A -85,B 0,C 180,E1 -14293.888,E2 -14293.888} C_VEL
LIN {X 0,Y 362.073,Z 441.774,A -85,B 0,C 180,E1 -14294.791,E2 -14294.791} C_VEL
LIN {X 0,Y 364.969,Z 444.311,A -85,B 0,C 180,E1 -14295.58,E2 -14295.58} C_VEL
LIN {X 0,Y 368.61,Z 448.162,A -85,B 0,C 180,E1 -14296.65,E2 -14296.65} C_VEL
LIN {X 0,Y 372.227,Z 451.023,A -85,B 0,C 180,E1 -14297.794,E2 -14297.794} C_VEL
LIN {X 0,Y 375.359,Z 454.327,A -85,B 0,C 180,E1 -14298.935,E2 -14298.935} C_VEL
LIN {X 0,Y 378.786,Z 456.802,A -85,B 0,C 180,E1 -14300.287,E2 -14300.287} C_VEL
LIN {X 0,Y 380.644,Z 458.067,A -85,B 0,C 180,E1 -14301.105,E2 -14301.105} C_VEL
LIN {X 0,Y 383.432,Z 461.255,A -85,B 0,C 180,E1 -14302.629,E2 -14302.629} C_VEL
LIN {X 0,Y 385.745,Z 463.129,A -85,B 0,C 180,E1 -14304.118,E2 -14304.118} C_VEL
LIN {X 0,Y 387.876,Z 464.258,A -85,B 0,C 180,E1 -14305.844,E2 -14305.844} C_VEL
LIN {X 0,Y 388.851,Z 464.488,A -85,B 0,C 180,E1 -14306.892,E2 -14306.892} C_VEL
LIN {X 0,Y 389.956,Z 464.674,A -85,B 0,C 180,E1 -14308.967,E2 -14308.967} C_VEL
LIN {X 0,Y 390.099,Z 464.734,A -85,B 0,C 180,E1 -14310,E2 -14310} C_VEL
LIN {X 0,Y 389.956,Z 464.673,A -85,B 0,C 180,E1 -14311.033,E2 -14311.033} C_VEL
LIN {X 0,Y 389.525,Z 464.665,A -85,B 0,C 180,E1 -14312.068,E2 -14312.068} C_VEL
LIN {X 0,Y 388.407,Z 464.375,A -85,B 0,C 180,E1 -14313.62,E2 -14313.62} C_VEL
LIN {X 0,Y 386.643,Z 463.695,A -85,B 0,C 180,E1 -14315.214,E2 -14315.214} C_VEL
LIN {X 0,Y 384.078,Z 461.854,A -85,B 0,C 180,E1 -14316.986,E2 -14316.986} C_VEL
LIN {X 0,Y 381.115,Z 458.702,A -85,B 0,C 180,E1 -14318.644,E2 -14318.644} C_VEL
LIN {X 0,Y 380.047,Z 457.474,A -85,B 0,C 180,E1 -14319.169,E2 -14319.169} C_VEL
LIN {X 0,Y 376.624,Z 455.342,A -85,B 0,C 180,E1 -14320.584,E2 -14320.584} C_VEL
LIN {X 0,Y 373.349,Z 452.345,A -85,B 0,C 180,E1 -14321.806,E2 -14321.806} C_VEL
LIN {X 0,Y 371.191,Z 450.074,A -85,B 0,C 180,E1 -14322.549,E2 -14322.549} C_VEL
LIN {X 0,Y 367.4,Z 447.023,A -85,B 0,C 180,E1 -14323.71,E2 -14323.71} C_VEL
LIN {X 0,Y 363.728,Z 443.069,A -85,B 0,C 180,E1 -14324.783,E2 -14324.783} C_VEL
LIN {X 0,Y 359.963,Z 439.642,A -85,B 0,C 180,E1 -14325.761,E2 -14325.761} C_VEL
LIN {X 0,Y 357.64,Z 436.878,A -85,B 0,C 180,E1 -14326.368,E2 -14326.368} C_VEL
LIN {X 0,Y 354.115,Z 433.359,A -85,B 0,C 180,E1 -14327.209,E2 -14327.209} C_VEL
LIN {X 0,Y 352.211,Z 430.967,A -85,B 0,C 180,E1 -14327.658,E2 -14327.658} C_VEL
LIN {X 0,Y 349.105,Z 427.563,A -85,B 0,C 180,E1 -14328.349,E2 -14328.349} C_VEL
LIN {X 0,Y 347.586,Z 425.439,A -85,B 0,C 180,E1 -14328.694,E2 -14328.694} C_VEL
LIN {X 0,Y 344.987,Z 422.505,A -85,B 0,C 180,E1 -14329.238,E2 -14329.238} C_VEL
LIN {X 0,Y 343.718,Z 420.461,A -85,B 0,C 180,E1 -14329.512,E2 -14329.512} C_VEL
LIN {X 0,Y 341.673,Z 418.195,A -85,B 0,C 180,E1 -14329.922,E2 -14329.922} C_VEL
LIN {X 0,Y 340.773,Z 415.537,A -85,B 0,C 180,E1 -14330.188,E2 -14330.188} C_VEL
LIN {X 0,Y 340.725,Z 415.542,A -85,B 0,C 180,E1 -14333.073,E2 -14333.073} C_VEL
LIN {X 0,Y 340.798,Z 415.532,A -85,B 0,C 180,E1 -14336.98,E2 -14336.98} C_VEL
LIN {X 0,Y 340.692,Z 415.546,A -85,B 0,C 180,E1 -14341.044,E2 -14341.044} C_VEL
LIN {X 0,Y 340.712,Z 415.546,A -85,B 0,C 180,E1 -14345.279,E2 -14345.279} C_VEL
LIN {X 0,Y 340.706,Z 415.542,A -85,B 0,C 180,E1 -14348.386,E2 -14348.386} C_VEL
LIN {X 0,Y 340.693,Z 415.544,A -85,B 0,C 180,E1 -14352.045,E2 -14352.045} C_VEL
LIN {X 0,Y 340.677,Z 415.55,A -85,B 0,C 180,E1 -14355.461,E2 -14355.461} C_VEL
LIN {X 0,Y 340.679,Z 415.547,A -85,B 0,C 180,E1 -14358.69,E2 -14358.69} C_VEL
LIN {X 0,Y 340.726,Z 415.54,A -85,B 0,C 180,E1 -14361.773,E2 -14361.773} C_VEL
LIN {X 0,Y 340.715,Z 415.542,A -85,B 0,C 180,E1 -14365.595,E2 -14365.595} C_VEL
LIN {X 0,Y 340.716,Z 415.541,A -85,B 0,C 180,E1 -14369.569,E2 -14369.569} C_VEL
LIN {X 0,Y 340.797,Z 415.536,A -85,B 0,C 180,E1 -14373.02,E2 -14373.02} C_VEL
LIN {X 0,Y 340.753,Z 415.537,A -85,B 0,C 180,E1 -14374.693,E2 -14374.693} C_VEL
LIN {X 0,Y 340.072,Z 415.624,A -85,B 0,C 180,E1 -14375.68,E2 -14375.68} C_VEL
LIN {X 0,Y 337.179,Z 415.984,A -85,B 0,C 180,E1 -14377.285,E2 -14377.285} C_VEL
LIN {X 0,Y 334.758,Z 416.286,A -85,B 0,C 180,E1 -14378.585,E2 -14378.585} C_VEL
LIN {X 0,Y 333.758,Z 416.407,A -85,B 0,C 180,E1 -14379.592,E2 -14379.592} C_VEL
LIN {X 0,Y 333.697,Z 416.414,A -85,B 0,C 180,E1 -14379.932,E2 -14379.932} C_VEL
LIN {X 0,Y 333.739,Z 416.415,A -85,B 0,C 180,E1 -14382.854,E2 -14382.854} C_VEL
LIN {X 0,Y 333.789,Z 416.407,A -85,B 0,C 180,E1 -14386.609,E2 -14386.609} C_VEL
LIN {X 0,Y 333.843,Z 416.399,A -85,B 0,C 180,E1 -14390.305,E2 -14390.305} C_VEL
LIN {X 0,Y 333.999,Z 416.382,A -85,B 0,C 180,E1 -14392.748,E2 -14392.748} C_VEL
LIN {X 0,Y 333.804,Z 416.402,A -85,B 0,C 180,E1 -14395.17,E2 -14395.17} C_VEL
LIN {X 0,Y 334.1,Z 416.361,A -85,B 0,C 180,E1 -14397.589,E2 -14397.589} C_VEL
LIN {X 0,Y 334.239,Z 416.346,A -85,B 0,C 180,E1 -14400.001,E2 -14400.001} C_VEL
LIN {X 0,Y 334.1,Z 416.369,A -85,B 0,C 180,E1 -14402.412,E2 -14402.412} C_VEL
LIN {X 0,Y 334.008,Z 416.379,A -85,B 0,C 180,E1 -14406.04,E2 -14406.04} C_VEL
LIN {X 0,Y 333.952,Z 416.389,A -85,B 0,C 180,E1 -14408.472,E2 -14408.472} C_VEL
LIN {X 0,Y 333.785,Z 416.409,A -85,B 0,C 180,E1 -14412.156,E2 -14412.156} C_VEL
LIN {X 0,Y 333.773,Z 416.408,A -85,B 0,C 180,E1 -14415.887,E2 -14415.887} C_VEL
LIN {X 0,Y 333.791,Z 416.406,A -85,B 0,C 180,E1 -14418.656,E2 -14418.656} C_VEL
LIN {X 0,Y 333.652,Z 416.426,A -85,B 0,C 180,E1 -14422.282,E2 -14422.282} C_VEL
LIN {X 0,Y 333.731,Z 416.416,A -85,B 0,C 180,E1 -14426.247,E2 -14426.247} C_VEL
LIN {X 0,Y 333.708,Z 416.415,A -85,B 0,C 180,E1 -14428.973,E2 -14428.973} C_VEL
LIN {X 0,Y 333.648,Z 416.425,A -85,B 0,C 180,E1 -14432.59,E2 -14432.59} C_VEL
LIN {X 0,Y 333.683,Z 416.422,A -85,B 0,C 180,E1 -14434.775,E2 -14434.775} C_VEL
LIN {X 0,Y 333.803,Z 417.445,A -85,B 0,C 180,E1 -14436.866,E2 -14436.866} C_VEL
LIN {X 0,Y 334.256,Z 420.375,A -85,B 0,C 180,E1 -14440.807,E2 -14440.807} C_VEL
LIN {X 0,Y 334.617,Z 423.276,A -85,B 0,C 180,E1 -14444.431,E2 -14444.431} C_VEL
LIN {X 0,Y 334.732,Z 426.275,A -85,B 0,C 180,E1 -14447.79,E2 -14447.79} C_VEL
LIN {X 0,Y 334.461,Z 429.411,A -85,B 0,C 180,E1 -14451.031,E2 -14451.031} C_VEL
LIN {X 0,Y 334.061,Z 432.376,A -85,B 0,C 180,E1 -14453.91,E2 -14453.91} C_VEL
LIN {X 0,Y 333.605,Z 436.164,A -85,B 0,C 180,E1 -14457.424,E2 -14457.424} C_VEL
LIN {X 0,Y 333.101,Z 440.166,A -85,B 0,C 180,E1 -14460.971,E2 -14460.971} C_VEL
LIN {X 0,Y 332.702,Z 444.924,A -85,B 0,C 180,E1 -14465.009,E2 -14465.009} C_VEL
LIN {X 0,Y 332.422,Z 448.909,A -85,B 0,C 180,E1 -14468.173,E2 -14468.173} C_VEL
LIN {X 0,Y 335.009,Z 459.9,A -85,B 0,C 180,E1 -14468.786,E2 -14468.786} C_VEL
LIN {X 0,Y 337.332,Z 472.264,A -85,B 0,C 180,E1 -14469.643,E2 -14469.643} C_VEL
LIN {X 0,Y 338.952,Z 485.271,A -85,B 0,C 180,E1 -14470.783,E2 -14470.783} C_VEL
LIN {X 0,Y 339.095,Z 490.186,A -85,B 0,C 180,E1 -14471.262,E2 -14471.262} C_VEL
LIN {X 0,Y 337.62,Z 502.375,A -85,B 0,C 180,E1 -14472.589,E2 -14472.589} C_VEL
LIN {X 0,Y 336.507,Z 511.3,A -85,B 0,C 180,E1 -14473.815,E2 -14473.815} C_VEL
LIN {X 0,Y 335.487,Z 519.26,A -85,B 0,C 180,E1 -14475.131,E2 -14475.131} C_VEL
LIN {X 0,Y 334.709,Z 525.464,A -85,B 0,C 180,E1 -14476.337,E2 -14476.337} C_VEL
LIN {X 0,Y 333.763,Z 531.999,A -85,B 0,C 180,E1 -14477.845,E2 -14477.845} C_VEL
LIN {X 0,Y 333.251,Z 536.503,A -85,B 0,C 180,E1 -14479.059,E2 -14479.059} C_VEL
LIN {X 0,Y 332.637,Z 541.996,A -85,B 0,C 180,E1 -14480.883,E2 -14480.883} C_VEL
LIN {X 0,Y 332.204,Z 546.321,A -85,B 0,C 180,E1 -14482.708,E2 -14482.708} C_VEL
LIN {X 0,Y 332.011,Z 549.116,A -85,B 0,C 180,E1 -14484.213,E2 -14484.213} C_VEL
LIN {X 0,Y 331.998,Z 551.88,A -85,B 0,C 180,E1 -14486.359,E2 -14486.359} C_VEL
LIN {X 0,Y 331.917,Z 552.937,A -85,B 0,C 180,E1 -14487.573,E2 -14487.573} C_VEL
LIN {X 0,Y 331.913,Z 553.526,A -85,B 0,C 180,E1 -14488.787,E2 -14488.787} C_VEL
LIN {X 0,Y 331.969,Z 553.682,A -85,B 0,C 180,E1 -14490,E2 -14490} C_VEL
LIN {X 0,Y 331.913,Z 553.526,A -85,B 0,C 180,E1 -14491.213,E2 -14491.213} C_VEL
LIN {X 0,Y 331.917,Z 552.937,A -85,B 0,C 180,E1 -14492.427,E2 -14492.427} C_VEL
LIN {X 0,Y 331.998,Z 551.88,A -85,B 0,C 180,E1 -14493.641,E2 -14493.641} C_VEL
LIN {X 0,Y 332.011,Z 549.116,A -85,B 0,C 180,E1 -14495.787,E2 -14495.787} C_VEL
LIN {X 0,Y 332.362,Z 545.081,A -85,B 0,C 180,E1 -14497.9,E2 -14497.9} C_VEL
LIN {X 0,Y 332.809,Z 540.335,A -85,B 0,C 180,E1 -14499.726,E2 -14499.726} C_VEL
LIN {X 0,Y 333.472,Z 534.311,A -85,B 0,C 180,E1 -14501.549,E2 -14501.549} C_VEL
LIN {X 0,Y 334.325,Z 528.215,A -85,B 0,C 180,E1 -14503.06,E2 -14503.06} C_VEL
LIN {X 0,Y 335.117,Z 522.516,A -85,B 0,C 180,E1 -14504.265,E2 -14504.265} C_VEL
LIN {X 0,Y 336.18,Z 513.96,A -85,B 0,C 180,E1 -14505.769,E2 -14505.769} C_VEL
LIN {X 0,Y 337.149,Z 505.778,A -85,B 0,C 180,E1 -14506.967,E2 -14506.967} C_VEL
LIN {X 0,Y 338.235,Z 497.268,A -85,B 0,C 180,E1 -14508.003,E2 -14508.003} C_VEL
LIN {X 0,Y 339.15,Z 488.551,A -85,B 0,C 180,E1 -14508.892,E2 -14508.892} C_VEL
LIN {X 0,Y 338.357,Z 479.801,A -85,B 0,C 180,E1 -14509.722,E2 -14509.722} C_VEL
LIN {X 0,Y 336.857,Z 469.575,A -85,B 0,C 180,E1 -14510.553,E2 -14510.553} C_VEL
LIN {X 0,Y 334.895,Z 459.279,A -85,B 0,C 180,E1 -14511.25,E2 -14511.25} C_VEL
LIN {X 0,Y 332.501,Z 449.531,A -85,B 0,C 180,E1 -14511.802,E2 -14511.802} C_VEL
LIN {X 0,Y 332.405,Z 448.649,A -85,B 0,C 180,E1 -14511.881,E2 -14511.881} C_VEL
LIN {X 0,Y 332.692,Z 444.892,A -85,B 0,C 180,E1 -14514.991,E2 -14514.991} C_VEL
LIN {X 0,Y 333.106,Z 440.162,A -85,B 0,C 180,E1 -14519.029,E2 -14519.029} C_VEL
LIN {X 0,Y 333.604,Z 436.157,A -85,B 0,C 180,E1 -14522.575,E2 -14522.575} C_VEL
LIN {X 0,Y 334.06,Z 432.368,A -85,B 0,C 180,E1 -14526.09,E2 -14526.09} C_VEL
LIN {X 0,Y 334.47,Z 429.303,A -85,B 0,C 180,E1 -14529.076,E2 -14529.076} C_VEL
LIN {X 0,Y 334.733,Z 426.253,A -85,B 0,C 180,E1 -14532.21,E2 -14532.21} C_VEL
LIN {X 0,Y 334.626,Z 423.275,A -85,B 0,C 180,E1 -14535.567,E2 -14535.567} C_VEL
LIN {X 0,Y 334.213,Z 420.213,A -85,B 0,C 180,E1 -14539.315,E2 -14539.315} C_VEL
LIN {X 0,Y 333.801,Z 417.445,A -85,B 0,C 180,E1 -14543.135,E2 -14543.135} C_VEL
LIN {X 0,Y 333.671,Z 416.427,A -85,B 0,C 180,E1 -14545.34,E2 -14545.34} C_VEL
LIN {X 0,Y 333.696,Z 416.42,A -85,B 0,C 180,E1 -14549.637,E2 -14549.637} C_VEL
LIN {X 0,Y 333.74,Z 416.412,A -85,B 0,C 180,E1 -14552.4,E2 -14552.4} C_VEL
LIN {X 0,Y 333.721,Z 416.413,A -85,B 0,C 180,E1 -14555.09,E2 -14555.09} C_VEL
LIN {X 0,Y 333.668,Z 416.419,A -85,B 0,C 180,E1 -14559.018,E2 -14559.018} C_VEL
LIN {X 0,Y 333.788,Z 416.408,A -85,B 0,C 180,E1 -14561.588,E2 -14561.588} C_VEL
LIN {X 0,Y 333.803,Z 416.407,A -85,B 0,C 180,E1 -14565.576,E2 -14565.576} C_VEL
LIN {X 0,Y 333.827,Z 416.4,A -85,B 0,C 180,E1 -14569.077,E2 -14569.077} C_VEL
LIN {X 0,Y 334,Z 416.377,A -85,B 0,C 180,E1 -14572.746,E2 -14572.746} C_VEL
LIN {X 0,Y 333.804,Z 416.404,A -85,B 0,C 180,E1 -14575.168,E2 -14575.168} C_VEL
LIN {X 0,Y 334.1,Z 416.369,A -85,B 0,C 180,E1 -14577.588,E2 -14577.588} C_VEL
LIN {X 0,Y 334.239,Z 416.346,A -85,B 0,C 180,E1 -14579.999,E2 -14579.999} C_VEL
LIN {X 0,Y 334.1,Z 416.361,A -85,B 0,C 180,E1 -14582.411,E2 -14582.411} C_VEL
LIN {X 0,Y 333.985,Z 416.38,A -85,B 0,C 180,E1 -14586.648,E2 -14586.648} C_VEL
LIN {X 0,Y 333.843,Z 416.399,A -85,B 0,C 180,E1 -14589.695,E2 -14589.695} C_VEL
LIN {X 0,Y 333.789,Z 416.407,A -85,B 0,C 180,E1 -14593.391,E2 -14593.391} C_VEL
LIN {X 0,Y 333.739,Z 416.415,A -85,B 0,C 180,E1 -14597.146,E2 -14597.146} C_VEL
LIN {X 0,Y 333.73,Z 416.411,A -85,B 0,C 180,E1 -14599.69,E2 -14599.69} C_VEL
LIN {X 0,Y 333.685,Z 416.417,A -85,B 0,C 180,E1 -14602.278,E2 -14602.278} C_VEL
LIN {X 0,Y 333.728,Z 416.411,A -85,B 0,C 180,E1 -14606.246,E2 -14606.246} C_VEL
LIN {X 0,Y 333.704,Z 416.42,A -85,B 0,C 180,E1 -14608.972,E2 -14608.972} C_VEL
LIN {X 0,Y 333.636,Z 416.425,A -85,B 0,C 180,E1 -14612.587,E2 -14612.587} C_VEL
LIN {X 0,Y 333.669,Z 416.419,A -85,B 0,C 180,E1 -14616.139,E2 -14616.139} C_VEL
LIN {X 0,Y 333.677,Z 416.42,A -85,B 0,C 180,E1 -14619.187,E2 -14619.187} C_VEL
LIN {X 0,Y 333.682,Z 416.42,A -85,B 0,C 180,E1 -14622.511,E2 -14622.511} C_VEL
LIN {X 0,Y 333.628,Z 416.424,A -85,B 0,C 180,E1 -14625.961,E2 -14625.961} C_VEL
LIN {X 0,Y 333.641,Z 416.423,A -85,B 0,C 180,E1 -14629.315,E2 -14629.315} C_VEL
LIN {X 0,Y 333.661,Z 416.421,A -85,B 0,C 180,E1 -14633.168,E2 -14633.168} C_VEL
LIN {X 0,Y 333.631,Z 416.427,A -85,B 0,C 180,E1 -14636.792,E2 -14636.792} C_VEL
LIN {X 0,Y 333.689,Z 416.417,A -85,B 0,C 180,E1 -14639.713,E2 -14639.713} C_VEL
LIN {X 0,Y 333.734,Z 416.416,A -85,B 0,C 180,E1 -14642.401,E2 -14642.401} C_VEL
LIN {X 0,Y 333.722,Z 416.414,A -85,B 0,C 180,E1 -14645.091,E2 -14645.091} C_VEL
LIN {X 0,Y 333.701,Z 416.49,A -85,B 0,C 180,E1 -14648.779,E2 -14648.779} C_VEL
LIN {X 0,Y 334.7,Z 419.303,A -85,B 0,C 180,E1 -14649.009,E2 -14649.009} C_VEL
LIN {X 0,Y 336.956,Z 421.968,A -85,B 0,C 180,E1 -14649.431,E2 -14649.431} C_VEL
LIN {X 0,Y 339.21,Z 425.265,A -85,B 0,C 180,E1 -14649.878,E2 -14649.878} C_VEL
LIN {X 0,Y 340.7,Z 426.974,A -85,B 0,C 180,E1 -14650.169,E2 -14650.169} C_VEL
LIN {X 0,Y 343.793,Z 430.836,A -85,B 0,C 180,E1 -14650.801,E2 -14650.801} C_VEL
LIN {X 0,Y 348.629,Z 436.473,A -85,B 0,C 180,E1 -14651.833,E2 -14651.833} C_VEL
LIN {X 0,Y 351.613,Z 439.84,A -85,B 0,C 180,E1 -14652.502,E2 -14652.502} C_VEL
LIN {X 0,Y 356.66,Z 444.991,A -85,B 0,C 180,E1 -14653.692,E2 -14653.692} C_VEL
LIN {X 0,Y 360.549,Z 448.877,A -85,B 0,C 180,E1 -14654.691,E2 -14654.691} C_VEL
LIN {X 0,Y 362.849,Z 450.955,A -85,B 0,C 180,E1 -14655.309,E2 -14655.309} C_VEL
LIN {X 0,Y 366.463,Z 454.695,A -85,B 0,C 180,E1 -14656.382,E2 -14656.382} C_VEL
LIN {X 0,Y 370.093,Z 457.6,A -85,B 0,C 180,E1 -14657.521,E2 -14657.521} C_VEL
LIN {X 0,Y 373.107,Z 460.763,A -85,B 0,C 180,E1 -14658.628,E2 -14658.628} C_VEL
LIN {X 0,Y 376.695,Z 463.395,A -85,B 0,C 180,E1 -14660.002,E2 -14660.002} C_VEL
LIN {X 0,Y 378.714,Z 464.716,A -85,B 0,C 180,E1 -14660.875,E2 -14660.875} C_VEL
LIN {X 0,Y 381.563,Z 467.972,A -85,B 0,C 180,E1 -14662.451,E2 -14662.451} C_VEL
LIN {X 0,Y 383.965,Z 469.949,A -85,B 0,C 180,E1 -14663.992,E2 -14663.992} C_VEL
LIN {X 0,Y 386.261,Z 471.147,A -85,B 0,C 180,E1 -14665.826,E2 -14665.826} C_VEL
LIN {X 0,Y 387.246,Z 471.404,A -85,B 0,C 180,E1 -14666.879,E2 -14666.879} C_VEL
LIN {X 0,Y 387.965,Z 471.522,A -85,B 0,C 180,E1 -14667.924,E2 -14667.924} C_VEL
LIN {X 0,Y 388.401,Z 471.601,A -85,B 0,C 180,E1 -14668.963,E2 -14668.963} C_VEL
LIN {X 0,Y 388.551,Z 471.663,A -85,B 0,C 180,E1 -14670,E2 -14670} C_VEL
LIN {X 0,Y 388.399,Z 471.597,A -85,B 0,C 180,E1 -14671.037,E2 -14671.037} C_VEL
LIN {X 0,Y 387.939,Z 471.581,A -85,B 0,C 180,E1 -14672.076,E2 -14672.076} C_VEL
LIN {X 0,Y 387.157,Z 471.351,A -85,B 0,C 180,E1 -14673.248,E2 -14673.248} C_VEL
LIN {X 0,Y 385.325,Z 470.759,A -85,B 0,C 180,E1 -14674.979,E2 -14674.979} C_VEL
LIN {X 0,Y 382.564,Z 468.925,A -85,B 0,C 180,E1 -14676.937,E2 -14676.937} C_VEL
LIN {X 0,Y 379.606,Z 465.887,A -85,B 0,C 180,E1 -14678.631,E2 -14678.631} C_VEL
LIN {X 0,Y 377.924,Z 464.116,A -85,B 0,C 180,E1 -14679.457,E2 -14679.457} C_VEL
LIN {X 0,Y 374.794,Z 462.165,A -85,B 0,C 180,E1 -14680.722,E2 -14680.722} C_VEL
LIN {X 0,Y 371.382,Z 459.084,A -85,B 0,C 180,E1 -14682.014,E2 -14682.014} C_VEL
LIN {X 0,Y 368.955,Z 456.551,A -85,B 0,C 180,E1 -14682.86,E2 -14682.86} C_VEL
LIN {X 0,Y 365.162,Z 453.493,A -85,B 0,C 180,E1 -14684.007,E2 -14684.007} C_VEL
LIN {X 0,Y 361.341,Z 449.449,A -85,B 0,C 180,E1 -14685.107,E2 -14685.107} C_VEL
LIN {X 0,Y 357.377,Z 445.829,A -85,B 0,C 180,E1 -14686.133,E2 -14686.133} C_VEL
